LIN {X 0,Y 282.332,Z 323.54,A -85,B 0,C 180,E1 -17008.574,E2 -17008.574} C_VEL
LIN {X 0,Y 282.332,Z 323.54,A -85,B 0,C 180,E1 -17011.426,E2 -17011.426} C_VEL
LIN {X 0,Y 282.337,Z 322.95,A -85,B 0,C 180,E1 -17012.854,E2 -17012.854} C_VEL
LIN {X 0,Y 282.388,Z 320.499,A -85,B 0,C 180,E1 -17015.713,E2 -17015.713} C_VEL
LIN {X 0,Y 282.677,Z 317.547,A -85,B 0,C 180,E1 -17017.859,E2 -17017.859} C_VEL
LIN {X 0,Y 283.169,Z 313.557,A -85,B 0,C 180,E1 -17020.005,E2 -17020.005} C_VEL
LIN {X 0,Y 283.939,Z 308.424,A -85,B 0,C 180,E1 -17022.145,E2 -17022.145} C_VEL
LIN {X 0,Y 284.955,Z 303.165,A -85,B 0,C 180,E1 -17023.914,E2 -17023.914} C_VEL
LIN {X 0,Y 286.081,Z 296.847,A -85,B 0,C 180,E1 -17025.678,E2 -17025.678} C_VEL
LIN {X 0,Y 287.264,Z 290.899,A -85,B 0,C 180,E1 -17027.073,E2 -17027.073} C_VEL
LIN {X 0,Y 288.4,Z 283.969,A -85,B 0,C 180,E1 -17028.469,E2 -17028.469} C_VEL
LIN {X 0,Y 289.834,Z 275.791,A -85,B 0,C 180,E1 -17029.845,E2 -17029.845} C_VEL
LIN {X 0,Y 291.272,Z 267.283,A -85,B 0,C 180,E1 -17031.033,E2 -17031.033} C_VEL
LIN {X 0,Y 292.592,Z 258.569,A -85,B 0,C 180,E1 -17032.043,E2 -17032.043} C_VEL
LIN {X 0,Y 293.904,Z 248.813,A -85,B 0,C 180,E1 -17032.959,E2 -17032.959} C_VEL
LIN {X 0,Y 294.936,Z 240.021,A -85,B 0,C 180,E1 -17033.617,E2 -17033.617} C_VEL
LIN {X 0,Y 295.878,Z 230.095,A -85,B 0,C 180,E1 -17034.188,E2 -17034.188} C_VEL
LIN {X 0,Y 296.511,Z 220.239,A -85,B 0,C 180,E1 -17034.599,E2 -17034.599} C_VEL
LIN {X 0,Y 297.245,Z 197.417,A -85,B 0,C 180,E1 -17035.188,E2 -17035.188} C_VEL
LIN {X 0,Y 298.174,Z 158.869,A -85,B 0,C 180,E1 -17036.112,E2 -17036.112} C_VEL
LIN {X 0,Y 294.383,Z 137.525,A -85,B 0,C 180,E1 -17037.041,E2 -17037.041} C_VEL
LIN {X 0,Y 290.06,Z 118.484,A -85,B 0,C 180,E1 -17037.995,E2 -17037.995} C_VEL
LIN {X 0,Y 288.045,Z 112.98,A -85,B 0,C 180,E1 -17038.403,E2 -17038.403} C_VEL
LIN {X 0,Y 287.272,Z 108.749,A -85,B 0,C 180,E1 -17040.101,E2 -17040.101} C_VEL
LIN {X 0,Y 285.619,Z 100.449,A -85,B 0,C 180,E1 -17043.786,E2 -17043.786} C_VEL
LIN {X 0,Y 284.383,Z 94.573,A -85,B 0,C 180,E1 -17046.598,E2 -17046.598} C_VEL
LIN {X 0,Y 284.309,Z 94.538,A -85,B 0,C 180,E1 -17049.994,E2 -17049.994} C_VEL
LIN {X 0,Y 284.248,Z 94.574,A -85,B 0,C 180,E1 -17054.19,E2 -17054.19} C_VEL
LIN {X 0,Y 284.274,Z 94.574,A -85,B 0,C 180,E1 -17058.124,E2 -17058.124} C_VEL
LIN {X 0,Y 284.324,Z 94.568,A -85,B 0,C 180,E1 -17062.277,E2 -17062.277} C_VEL
LIN {X 0,Y 284.31,Z 94.547,A -85,B 0,C 180,E1 -17065.35,E2 -17065.35} C_VEL
LIN {X 0,Y 284.295,Z 94.571,A -85,B 0,C 180,E1 -17068.725,E2 -17068.725} C_VEL
LIN {X 0,Y 284.396,Z 94.53,A -85,B 0,C 180,E1 -17072.827,E2 -17072.827} C_VEL
LIN {X 0,Y 284.368,Z 94.562,A -85,B 0,C 180,E1 -17076.706,E2 -17076.706} C_VEL
LIN {X 0,Y 284.404,Z 94.52,A -85,B 0,C 180,E1 -17081.261,E2 -17081.261} C_VEL
LIN {X 0,Y 284.493,Z 94.54,A -85,B 0,C 180,E1 -17084.458,E2 -17084.458} C_VEL
LIN {X 0,Y 284.489,Z 94.522,A -85,B 0,C 180,E1 -17088.601,E2 -17088.601} C_VEL
LIN {X 0,Y 284.66,Z 94.494,A -85,B 0,C 180,E1 -17091.48,E2 -17091.48} C_VEL
LIN {X 0,Y 284.603,Z 94.533,A -85,B 0,C 180,E1 -17094.331,E2 -17094.331} C_VEL
LIN {X 0,Y 284.854,Z 94.474,A -85,B 0,C 180,E1 -17098.585,E2 -17098.585} C_VEL
LIN {X 0,Y 284.854,Z 94.471,A -85,B 0,C 180,E1 -17101.413,E2 -17101.413} C_VEL
LIN {X 0,Y 284.698,Z 94.51,A -85,B 0,C 180,E1 -17107.089,E2 -17107.089} C_VEL
LIN {X 0,Y 284.566,Z 94.499,A -85,B 0,C 180,E1 -17109.955,E2 -17109.955} C_VEL
LIN {X 0,Y 284.481,Z 94.548,A -85,B 0,C 180,E1 -17114.302,E2 -17114.302} C_VEL
LIN {X 0,Y 284.424,Z 94.535,A -85,B 0,C 180,E1 -17117.248,E2 -17117.248} C_VEL
LIN {X 0,Y 284.377,Z 94.535,A -85,B 0,C 180,E1 -17120.241,E2 -17120.241} C_VEL
LIN {X 0,Y 284.368,Z 94.561,A -85,B 0,C 180,E1 -17123.875,E2 -17123.875} C_VEL
LIN {X 0,Y 284.393,Z 94.532,A -85,B 0,C 180,E1 -17127.172,E2 -17127.172} C_VEL
LIN {X 0,Y 284.291,Z 94.573,A -85,B 0,C 180,E1 -17131.274,E2 -17131.274} C_VEL
LIN {X 0,Y 284.359,Z 94.546,A -85,B 0,C 180,E1 -17135.353,E2 -17135.353} C_VEL
LIN {X 0,Y 284.327,Z 94.57,A -85,B 0,C 180,E1 -17138.166,E2 -17138.166} C_VEL
LIN {X 0,Y 284.289,Z 94.564,A -85,B 0,C 180,E1 -17141.871,E2 -17141.871} C_VEL
LIN {X 0,Y 284.251,Z 94.537,A -85,B 0,C 180,E1 -17146.189,E2 -17146.189} C_VEL
LIN {X 0,Y 284.304,Z 94.538,A -85,B 0,C 180,E1 -17150.023,E2 -17150.023} C_VEL
LIN {X 0,Y 284.346,Z 94.545,A -85,B 0,C 180,E1 -17153.616,E2 -17153.616} C_VEL
LIN {X 0,Y 284.304,Z 94.553,A -85,B 0,C 180,E1 -17157.189,E2 -17157.189} C_VEL
LIN {X 0,Y 284.358,Z 94.704,A -85,B 0,C 180,E1 -17160.852,E2 -17160.852} C_VEL
LIN {X 0,Y 284.571,Z 95.611,A -85,B 0,C 180,E1 -17161.125,E2 -17161.125} C_VEL
LIN {X 0,Y 292.908,Z 111.214,A -85,B 0,C 180,E1 -17162.479,E2 -17162.479} C_VEL
LIN {X 0,Y 301.128,Z 122.682,A -85,B 0,C 180,E1 -17163.597,E2 -17163.597} C_VEL
LIN {X 0,Y 308.763,Z 131.233,A -85,B 0,C 180,E1 -17164.598,E2 -17164.598} C_VEL
LIN {X 0,Y 315.019,Z 137.865,A -85,B 0,C 180,E1 -17165.516,E2 -17165.516} C_VEL
LIN {X 0,Y 321.23,Z 144.234,A -85,B 0,C 180,E1 -17166.527,E2 -17166.527} C_VEL
LIN {X 0,Y 328.563,Z 151.312,A -85,B 0,C 180,E1 -17167.868,E2 -17167.868} C_VEL
LIN {X 0,Y 335.56,Z 157.924,A -85,B 0,C 180,E1 -17169.294,E2 -17169.294} C_VEL
LIN {X 0,Y 343.832,Z 165.121,A -85,B 0,C 180,E1 -17171.117,E2 -17171.117} C_VEL
LIN {X 0,Y 349.126,Z 169.383,A -85,B 0,C 180,E1 -17172.401,E2 -17172.401} C_VEL
LIN {X 0,Y 354.265,Z 173.621,A -85,B 0,C 180,E1 -17173.763,E2 -17173.763} C_VEL
LIN {X 0,Y 359.027,Z 177.249,A -85,B 0,C 180,E1 -17175.137,E2 -17175.137} C_VEL
LIN {X 0,Y 363.782,Z 181.091,A -85,B 0,C 180,E1 -17176.663,E2 -17176.663} C_VEL
LIN {X 0,Y 368.414,Z 183.996,A -85,B 0,C 180,E1 -17178.318,E2 -17178.318} C_VEL
LIN {X 0,Y 370.691,Z 185.609,A -85,B 0,C 180,E1 -17179.249,E2 -17179.249} C_VEL
LIN {X 0,Y 374.324,Z 188.697,A -85,B 0,C 180,E1 -17180.953,E2 -17180.953} C_VEL
LIN {X 0,Y 377.385,Z 190.784,A -85,B 0,C 180,E1 -17182.671,E2 -17182.671} C_VEL
LIN {X 0,Y 379.747,Z 192.052,A -85,B 0,C 180,E1 -17184.313,E2 -17184.313} C_VEL
LIN {X 0,Y 381.337,Z 192.728,A -85,B 0,C 180,E1 -17185.772,E2 -17185.772} C_VEL
LIN {X 0,Y 382.556,Z 193.147,A -85,B 0,C 180,E1 -17187.355,E2 -17187.355} C_VEL
LIN {X 0,Y 383.205,Z 193.6,A -85,B 0,C 180,E1 -17188.949,E2 -17188.949} C_VEL
LIN {X 0,Y 383.351,Z 193.507,A -85,B 0,C 180,E1 -17190,E2 -17190} C_VEL
LIN {X 0,Y 383.05,Z 193.43,A -85,B 0,C 180,E1 -17191.577,E2 -17191.577} C_VEL
LIN {X 0,Y 382.228,Z 192.953,A -85,B 0,C 180,E1 -17193.162,E2 -17193.162} C_VEL
LIN {X 0,Y 380.501,Z 192.419,A -85,B 0,C 180,E1 -17195.024,E2 -17195.024} C_VEL
LIN {X 0,Y 377.946,Z 191.113,A -85,B 0,C 180,E1 -17196.961,E2 -17196.961} C_VEL
LIN {X 0,Y 374.627,Z 188.924,A -85,B 0,C 180,E1 -17198.885,E2 -17198.885} C_VEL
LIN {X 0,Y 371.12,Z 186.009,A -85,B 0,C 180,E1 -17200.562,E2 -17200.562} C_VEL
LIN {X 0,Y 369.133,Z 184.402,A -85,B 0,C 180,E1 -17201.397,E2 -17201.397} C_VEL
LIN {X 0,Y 364.42,Z 181.507,A -85,B 0,C 180,E1 -17203.127,E2 -17203.127} C_VEL
LIN {X 0,Y 359.32,Z 177.506,A -85,B 0,C 180,E1 -17204.77,E2 -17204.77} C_VEL
LIN {X 0,Y 355.345,Z 174.403,A -85,B 0,C 180,E1 -17205.935,E2 -17205.935} C_VEL
LIN {X 0,Y 349.645,Z 169.914,A -85,B 0,C 180,E1 -17207.46,E2 -17207.46} C_VEL
LIN {X 0,Y 345.087,Z 166.059,A -85,B 0,C 180,E1 -17208.584,E2 -17208.584} C_VEL
LIN {X 0,Y 339.388,Z 161.216,A -85,B 0,C 180,E1 -17209.892,E2 -17209.892} C_VEL
LIN {X 0,Y 331.39,Z 154.073,A -85,B 0,C 180,E1 -17211.572,E2 -17211.572} C_VEL
LIN {X 0,Y 323.333,Z 146.328,A -85,B 0,C 180,E1 -17213.097,E2 -17213.097} C_VEL
LIN {X 0,Y 316.271,Z 139.268,A -85,B 0,C 180,E1 -17214.282,E2 -17214.282} C_VEL
LIN {X 0,Y 307.947,Z 130.457,A -85,B 0,C 180,E1 -17215.508,E2 -17215.508} C_VEL
LIN {X 0,Y 299.459,Z 120.55,A -85,B 0,C 180,E1 -17216.619,E2 -17216.619} C_VEL
LIN {X 0,Y 292.1,Z 109.823,A -85,B 0,C 180,E1 -17217.642,E2 -17217.642} C_VEL
LIN {X 0,Y 284.572,Z 95.609,A -85,B 0,C 180,E1 -17218.876,E2 -17218.876} C_VEL
LIN {X 0,Y 284.349,Z 94.626,A -85,B 0,C 180,E1 -17219.19,E2 -17219.19} C_VEL
LIN {X 0,Y 284.302,Z 94.55,A -85,B 0,C 180,E1 -17222.946,E2 -17222.946} C_VEL
LIN {X 0,Y 284.346,Z 94.544,A -85,B 0,C 180,E1 -17226.384,E2 -17226.384} C_VEL
LIN {X 0,Y 284.303,Z 94.538,A -85,B 0,C 180,E1 -17229.995,E2 -17229.995} C_VEL
LIN {X 0,Y 284.241,Z 94.546,A -85,B 0,C 180,E1 -17234.191,E2 -17234.191} C_VEL
LIN {X 0,Y 284.289,Z 94.564,A -85,B 0,C 180,E1 -17238.129,E2 -17238.129} C_VEL
LIN {X 0,Y 284.327,Z 94.57,A -85,B 0,C 180,E1 -17241.834,E2 -17241.834} C_VEL
LIN {X 0,Y 284.321,Z 94.547,A -85,B 0,C 180,E1 -17245.353,E2 -17245.353} C_VEL
LIN {X 0,Y 284.291,Z 94.573,A -85,B 0,C 180,E1 -17248.726,E2 -17248.726} C_VEL
LIN {X 0,Y 284.393,Z 94.532,A -85,B 0,C 180,E1 -17252.828,E2 -17252.828} C_VEL
LIN {X 0,Y 284.365,Z 94.565,A -85,B 0,C 180,E1 -17256.708,E2 -17256.708} C_VEL
LIN {X 0,Y 284.401,Z 94.525,A -85,B 0,C 180,E1 -17261.262,E2 -17261.262} C_VEL
LIN {X 0,Y 284.491,Z 94.544,A -85,B 0,C 180,E1 -17264.46,E2 -17264.46} C_VEL
LIN {X 0,Y 284.489,Z 94.522,A -85,B 0,C 180,E1 -17268.602,E2 -17268.602} C_VEL
LIN {X 0,Y 284.658,Z 94.497,A -85,B 0,C 180,E1 -17271.482,E2 -17271.482} C_VEL
LIN {X 0,Y 284.601,Z 94.533,A -85,B 0,C 180,E1 -17274.332,E2 -17274.332} C_VEL
LIN {X 0,Y 284.854,Z 94.471,A -85,B 0,C 180,E1 -17278.587,E2 -17278.587} C_VEL
LIN {X 0,Y 284.854,Z 94.474,A -85,B 0,C 180,E1 -17281.415,E2 -17281.415} C_VEL
LIN {X 0,Y 284.7,Z 94.508,A -85,B 0,C 180,E1 -17287.091,E2 -17287.091} C_VEL
LIN {X 0,Y 284.567,Z 94.498,A -85,B 0,C 180,E1 -17289.956,E2 -17289.956} C_VEL
LIN {X 0,Y 284.483,Z 94.545,A -85,B 0,C 180,E1 -17294.303,E2 -17294.303} C_VEL
LIN {X 0,Y 284.426,Z 94.529,A -85,B 0,C 180,E1 -17297.249,E2 -17297.249} C_VEL
LIN {X 0,Y 284.384,Z 94.531,A -85,B 0,C 180,E1 -17299.999,E2 -17299.999} C_VEL
LIN {X 0,Y 283.746,Z 94.627,A -85,B 0,C 180,E1 -17301.182,E2 -17301.182} C_VEL
LIN {X 0,Y 280.868,Z 94.998,A -85,B 0,C 180,E1 -17303.108,E2 -17303.108} C_VEL
LIN {X 0,Y 278.417,Z 95.294,A -85,B 0,C 180,E1 -17304.672,E2 -17304.672} C_VEL
LIN {X 0,Y 277.381,Z 95.409,A -85,B 0,C 180,E1 -17305.885,E2 -17305.885} C_VEL
LIN {X 0,Y 277.308,Z 95.414,A -85,B 0,C 180,E1 -17306.296,E2 -17306.296} C_VEL
LIN {X 0,Y 277.274,Z 95.446,A -85,B 0,C 180,E1 -17310.482,E2 -17310.482} C_VEL
LIN {X 0,Y 277.248,Z 95.426,A -85,B 0,C 180,E1 -17313.896,E2 -17313.896} C_VEL
LIN {X 0,Y 277.27,Z 95.447,A -85,B 0,C 180,E1 -17317.47,E2 -17317.47} C_VEL
LIN {X 0,Y 277.212,Z 95.444,A -85,B 0,C 180,E1 -17321.237,E2 -17321.237} C_VEL
LIN {X 0,Y 277.203,Z 95.446,A -85,B 0,C 180,E1 -17325.227,E2 -17325.227} C_VEL
LIN {X 0,Y 277.225,Z 95.42,A -85,B 0,C 180,E1 -17329.513,E2 -17329.513} C_VEL
LIN {X 0,Y 277.341,Z 95.56,A -85,B 0,C 180,E1 -17332.959,E2 -17332.959} C_VEL
LIN {X 0,Y 278.814,Z 102.621,A -85,B 0,C 180,E1 -17336.32,E2 -17336.32} C_VEL
LIN {X 0,Y 280.364,Z 110.466,A -85,B 0,C 180,E1 -17339.911,E2 -17339.911} C_VEL
LIN {X 0,Y 280.827,Z 112.758,A -85,B 0,C 180,E1 -17340.794,E2 -17340.794} C_VEL
LIN {X 0,Y 284.469,Z 122.35,A -85,B 0,C 180,E1 -17341.518,E2 -17341.518} C_VEL
LIN {X 0,Y 289.627,Z 146.77,A -85,B 0,C 180,E1 -17342.734,E2 -17342.734} C_VEL
LIN {X 0,Y 291.872,Z 160.971,A -85,B 0,C 180,E1 -17343.342,E2 -17343.342} C_VEL
LIN {X 0,Y 290.223,Z 218.73,A -85,B 0,C 180,E1 -17344.783,E2 -17344.783} C_VEL
LIN {X 0,Y 289.49,Z 229.031,A -85,B 0,C 180,E1 -17345.195,E2 -17345.195} C_VEL
LIN {X 0,Y 288.543,Z 238.542,A -85,B 0,C 180,E1 -17345.731,E2 -17345.731} C_VEL
LIN {X 0,Y 287.418,Z 248.624,A -85,B 0,C 180,E1 -17346.492,E2 -17346.492} C_VEL
LIN {X 0,Y 286.034,Z 258.379,A -85,B 0,C 180,E1 -17347.424,E2 -17347.424} C_VEL
LIN {X 0,Y 284.398,Z 268.442,A -85,B 0,C 180,E1 -17348.623,E2 -17348.623} C_VEL
LIN {X 0,Y 282.361,Z 279.94,A -85,B 0,C 180,E1 -17350.366,E2 -17350.366} C_VEL
LIN {X 0,Y 280.716,Z 288.731,A -85,B 0,C 180,E1 -17352.06,E2 -17352.06} C_VEL
LIN {X 0,Y 279.503,Z 295.28,A -85,B 0,C 180,E1 -17353.568,E2 -17353.568} C_VEL
LIN {X 0,Y 278.263,Z 301.818,A -85,B 0,C 180,E1 -17355.371,E2 -17355.371} C_VEL
LIN {X 0,Y 277.338,Z 306.317,A -85,B 0,C 180,E1 -17356.817,E2 -17356.817} C_VEL
LIN {X 0,Y 276.386,Z 311.811,A -85,B 0,C 180,E1 -17359.006,E2 -17359.006} C_VEL
LIN {X 0,Y 275.745,Z 316.138,A -85,B 0,C 180,E1 -17361.204,E2 -17361.204} C_VEL
LIN {X 0,Y 275.496,Z 318.507,A -85,B 0,C 180,E1 -17362.672,E2 -17362.672} C_VEL
LIN {X 0,Y 275.249,Z 321,A -85,B 0,C 180,E1 -17364.751,E2 -17364.751} C_VEL
LIN {X 0,Y 275.246,Z 322.759,A -85,B 0,C 180,E1 -17367.073,E2 -17367.073} C_VEL
LIN {X 0,Y 275.256,Z 323.35,A -85,B 0,C 180,E1 -17368.537,E2 -17368.537} C_VEL
LIN {X 0,Y 275.256,Z 323.35,A -85,B 0,C 180,E1 -17371.463,E2 -17371.463} C_VEL
LIN {X 0,Y 275.246,Z 322.759,A -85,B 0,C 180,E1 -17372.927,E2 -17372.927} C_VEL
LIN {X 0,Y 275.302,Z 320.308,A -85,B 0,C 180,E1 -17375.861,E2 -17375.861} C_VEL
LIN {X 0,Y 275.606,Z 317.356,A -85,B 0,C 180,E1 -17378.062,E2 -17378.062} C_VEL
LIN {X 0,Y 276.159,Z 313.366,A -85,B 0,C 180,E1 -17380.262,E2 -17380.262} C_VEL
LIN {X 0,Y 276.965,Z 308.233,A -85,B 0,C 180,E1 -17382.456,E2 -17382.456} C_VEL
LIN {X 0,Y 278.02,Z 302.973,A -85,B 0,C 180,E1 -17384.269,E2 -17384.269} C_VEL
LIN {X 0,Y 279.218,Z 296.655,A -85,B 0,C 180,E1 -17386.074,E2 -17386.074} C_VEL
LIN {X 0,Y 280.673,Z 289.683,A -85,B 0,C 180,E1 -17387.723,E2 -17387.723} C_VEL
LIN {X 0,Y 281.661,Z 283.778,A -85,B 0,C 180,E1 -17388.928,E2 -17388.928} C_VEL
LIN {X 0,Y 283.156,Z 275.601,A -85,B 0,C 180,E1 -17390.333,E2 -17390.333} C_VEL
LIN {X 0,Y 284.652,Z 267.092,A -85,B 0,C 180,E1 -17391.547,E2 -17391.547} C_VEL
LIN {X 0,Y 286.016,Z 258.378,A -85,B 0,C 180,E1 -17392.578,E2 -17392.578} C_VEL
LIN {X 0,Y 287.379,Z 248.622,A -85,B 0,C 180,E1 -17393.511,E2 -17393.511} C_VEL
LIN {X 0,Y 288.438,Z 239.831,A -85,B 0,C 180,E1 -17394.183,E2 -17394.183} C_VEL
LIN {X 0,Y 289.418,Z 229.905,A -85,B 0,C 180,E1 -17394.764,E2 -17394.764} C_VEL
LIN {X 0,Y 290.084,Z 220.049,A -85,B 0,C 180,E1 -17395.182,E2 -17395.182} C_VEL
LIN {X 0,Y 290.824,Z 197.226,A -85,B 0,C 180,E1 -17395.784,E2 -17395.784} C_VEL
LIN {X 0,Y 291.8,Z 159.943,A -85,B 0,C 180,E1 -17396.693,E2 -17396.693} C_VEL
LIN {X 0,Y 288.2,Z 139.453,A -85,B 0,C 180,E1 -17397.612,E2 -17397.612} C_VEL
LIN {X 0,Y 284.11,Z 121.147,A -85,B 0,C 180,E1 -17398.555,E2 -17398.555} C_VEL
LIN {X 0,Y 280.821,Z 112.765,A -85,B 0,C 180,E1 -17399.203,E2 -17399.203} C_VEL
LIN {X 0,Y 280.099,Z 109.079,A -85,B 0,C 180,E1 -17400.721,E2 -17400.721} C_VEL
LIN {X 0,Y 278.839,Z 102.522,A -85,B 0,C 180,E1 -17403.72,E2 -17403.72} C_VEL
LIN {X 0,Y 277.342,Z 95.462,A -85,B 0,C 180,E1 -17407.144,E2 -17407.144} C_VEL
LIN {X 0,Y 277.212,Z 95.428,A -85,B 0,C 180,E1 -17411.236,E2 -17411.236} C_VEL
LIN {X 0,Y 277.203,Z 95.446,A -85,B 0,C 180,E1 -17415.226,E2 -17415.226} C_VEL
LIN {X 0,Y 277.224,Z 95.437,A -85,B 0,C 180,E1 -17419.512,E2 -17419.512} C_VEL
LIN {X 0,Y 277.27,Z 95.447,A -85,B 0,C 180,E1 -17422.53,E2 -17422.53} C_VEL
LIN {X 0,Y 277.248,Z 95.426,A -85,B 0,C 180,E1 -17426.104,E2 -17426.104} C_VEL
LIN {X 0,Y 277.263,Z 95.447,A -85,B 0,C 180,E1 -17429.538,E2 -17429.538} C_VEL
LIN {X 0,Y 277.358,Z 95.406,A -85,B 0,C 180,E1 -17432.863,E2 -17432.863} C_VEL
LIN {X 0,Y 277.33,Z 95.435,A -85,B 0,C 180,E1 -17436.079,E2 -17436.079} C_VEL
LIN {X 0,Y 277.346,Z 95.4,A -85,B 0,C 180,E1 -17440.765,E2 -17440.765} C_VEL
LIN {X 0,Y 277.436,Z 95.423,A -85,B 0,C 180,E1 -17445.325,E2 -17445.325} C_VEL
LIN {X 0,Y 277.507,Z 95.378,A -85,B 0,C 180,E1 -17449.788,E2 -17449.788} C_VEL
LIN {X 0,Y 277.655,Z 95.382,A -85,B 0,C 180,E1 -17452.728,E2 -17452.728} C_VEL
LIN {X 0,Y 277.82,Z 95.35,A -85,B 0,C 180,E1 -17458.55,E2 -17458.55} C_VEL
LIN {X 0,Y 277.82,Z 95.347,A -85,B 0,C 180,E1 -17461.449,E2 -17461.449} C_VEL
LIN {X 0,Y 277.653,Z 95.384,A -85,B 0,C 180,E1 -17467.27,E2 -17467.27} C_VEL
LIN {X 0,Y 277.507,Z 95.379,A -85,B 0,C 180,E1 -17470.21,E2 -17470.21} C_VEL
LIN {X 0,Y 277.434,Z 95.426,A -85,B 0,C 180,E1 -17474.673,E2 -17474.673} C_VEL
LIN {X 0,Y 277.343,Z 95.403,A -85,B 0,C 180,E1 -17479.233,E2 -17479.233} C_VEL
LIN {X 0,Y 277.318,Z 95.439,A -85,B 0,C 180,E1 -17484.17,E2 -17484.17} C_VEL
LIN {X 0,Y 277.321,Z 95.412,A -85,B 0,C 180,E1 -17487.504,E2 -17487.504} C_VEL
LIN {X 0,Y 277.27,Z 95.446,A -85,B 0,C 180,E1 -17490.481,E2 -17490.481} C_VEL
LIN {X 0,Y 277.251,Z 95.428,A -85,B 0,C 180,E1 -17493.894,E2 -17493.894} C_VEL
LIN {X 0,Y 277.283,Z 95.447,A -85,B 0,C 180,E1 -17497.466,E2 -17497.466} C_VEL
LIN {X 0,Y 277.231,Z 95.436,A -85,B 0,C 180,E1 -17501.232,E2 -17501.232} C_VEL
LIN {X 0,Y 277.2,Z 95.434,A -85,B 0,C 180,E1 -17505.225,E2 -17505.225} C_VEL
LIN {X 0,Y 277.218,Z 95.409,A -85,B 0,C 180,E1 -17509.512,E2 -17509.512} C_VEL
LIN {X 0,Y 277.278,Z 95.445,A -85,B 0,C 180,E1 -17512.533,E2 -17512.533} C_VEL
LIN {X 0,Y 277.25,Z 95.415,A -85,B 0,C 180,E1 -17516.105,E2 -17516.105} C_VEL
LIN {X 0,Y 277.307,Z 95.57,A -85,B 0,C 180,E1 -17520.071,E2 -17520.071} C_VEL
LIN {X 0,Y 277.558,Z 96.523,A -85,B 0,C 180,E1 -17520.347,E2 -17520.347} C_VEL
LIN {X 0,Y 287.675,Z 115.487,A -85,B 0,C 180,E1 -17522.049,E2 -17522.049} C_VEL
LIN {X 0,Y 296.033,Z 127.245,A -85,B 0,C 180,E1 -17523.224,E2 -17523.224} C_VEL
LIN {X 0,Y 304.437,Z 136.633,A -85,B 0,C 180,E1 -17524.285,E2 -17524.285} C_VEL
LIN {X 0,Y 311.55,Z 144.001,A -85,B 0,C 180,E1 -17525.264,E2 -17525.264} C_VEL
LIN {X 0,Y 317.642,Z 150.071,A -85,B 0,C 180,E1 -17526.194,E2 -17526.194} C_VEL
LIN {X 0,Y 324.32,Z 156.446,A -85,B 0,C 180,E1 -17527.349,E2 -17527.349} C_VEL
LIN {X 0,Y 332.199,Z 163.7,A -85,B 0,C 180,E1 -17528.859,E2 -17528.859} C_VEL
LIN {X 0,Y 340.746,Z 171.076,A -85,B 0,C 180,E1 -17530.692,E2 -17530.692} C_VEL
LIN {X 0,Y 346.717,Z 175.77,A -85,B 0,C 180,E1 -17532.086,E2 -17532.086} C_VEL
LIN {X 0,Y 352.189,Z 180.199,A -85,B 0,C 180,E1 -17533.491,E2 -17533.491} C_VEL
LIN {X 0,Y 357.449,Z 184.156,A -85,B 0,C 180,E1 -17534.97,E2 -17534.97} C_VEL
LIN {X 0,Y 362.886,Z 188.383,A -85,B 0,C 180,E1 -17536.697,E2 -17536.697} C_VEL
LIN {X 0,Y 367.765,Z 191.274,A -85,B 0,C 180,E1 -17538.433,E2 -17538.433} C_VEL
LIN {X 0,Y 372.315,Z 195.056,A -85,B 0,C 180,E1 -17540.433,E2 -17540.433} C_VEL
LIN {X 0,Y 375.651,Z 197.365,A -85,B 0,C 180,E1 -17542.185,E2 -17542.185} C_VEL
LIN {X 0,Y 378.536,Z 198.953,A -85,B 0,C 180,E1 -17544.075,E2 -17544.075} C_VEL
LIN {X 0,Y 380.515,Z 199.785,A -85,B 0,C 180,E1 -17545.828,E2 -17545.828} C_VEL
LIN {X 0,Y 381.686,Z 200.194,A -85,B 0,C 180,E1 -17547.349,E2 -17547.349} C_VEL
LIN {X 0,Y 382.34,Z 200.646,A -85,B 0,C 180,E1 -17548.947,E2 -17548.947} C_VEL
LIN {X 0,Y 382.488,Z 200.539,A -85,B 0,C 180,E1 -17550,E2 -17550} C_VEL
LIN {X 0,Y 382.181,Z 200.478,A -85,B 0,C 180,E1 -17551.581,E2 -17551.581} C_VEL
LIN {X 0,Y 381.092,Z 199.929,A -85,B 0,C 180,E1 -17553.513,E2 -17553.513} C_VEL
LIN {X 0,Y 379.107,Z 199.217,A -85,B 0,C 180,E1 -17555.477,E2 -17555.477} C_VEL
LIN {X 0,Y 376.465,Z 197.808,A -85,B 0,C 180,E1 -17557.348,E2 -17557.348} C_VEL
LIN {X 0,Y 373.181,Z 195.688,A -85,B 0,C 180,E1 -17559.153,E2 -17559.153} C_VEL
LIN {X 0,Y 369.493,Z 192.66,A -85,B 0,C 180,E1 -17560.852,E2 -17560.852} C_VEL
LIN {X 0,Y 367.139,Z 190.928,A -85,B 0,C 180,E1 -17561.798,E2 -17561.798} C_VEL
LIN {X 0,Y 362.576,Z 188.136,A -85,B 0,C 180,E1 -17563.407,E2 -17563.407} C_VEL
LIN {X 0,Y 357.452,Z 184.132,A -85,B 0,C 180,E1 -17565.03,E2 -17565.03} C_VEL
LIN {X 0,Y 351.476,Z 179.651,A -85,B 0,C 180,E1 -17566.701,E2 -17566.701} C_VEL
LIN {X 0,Y 345.974,Z 175.162,A -85,B 0,C 180,E1 -17568.096,E2 -17568.096} C_VEL
LIN {X 0,Y 337.981,Z 168.729,A -85,B 0,C 180,E1 -17569.928,E2 -17569.928} C_VEL
LIN {X 0,Y 329.178,Z 160.994,A -85,B 0,C 180,E1 -17571.739,E2 -17571.739} C_VEL
LIN {X 0,Y 320.365,Z 152.707,A -85,B 0,C 180,E1 -17573.351,E2 -17573.351} C_VEL
LIN {X 0,Y 312.398,Z 144.958,A -85,B 0,C 180,E1 -17574.611,E2 -17574.611} C_VEL
LIN {X 0,Y 303.796,Z 136.018,A -85,B 0,C 180,E1 -17575.795,E2 -17575.795} C_VEL
LIN {X 0,Y 294.334,Z 125.049,A -85,B 0,C 180,E1 -17577.003,E2 -17577.003} C_VEL
LIN {X 0,Y 287.007,Z 114.312,A -85,B 0,C 180,E1 -17578.055,E2 -17578.055} C_VEL
LIN {X 0,Y 277.551,Z 96.544,A -85,B 0,C 180,E1 -17579.65,E2 -17579.65} C_VEL
LIN {X 0,Y 277.302,Z 95.517,A -85,B 0,C 180,E1 -17579.965,E2 -17579.965} C_VEL
LIN {X 0,Y 277.251,Z 95.415,A -85,B 0,C 180,E1 -17583.895,E2 -17583.895} C_VEL
LIN {X 0,Y 277.278,Z 95.445,A -85,B 0,C 180,E1 -17587.467,E2 -17587.467} C_VEL
LIN {X 0,Y 277.206,Z 95.401,A -85,B 0,C 180,E1 -17591.237,E2 -17591.237} C_VEL
LIN {X 0,Y 277.204,Z 95.445,A -85,B 0,C 180,E1 -17595.226,E2 -17595.226} C_VEL
LIN {X 0,Y 277.257,Z 95.431,A -85,B 0,C 180,E1 -17599.504,E2 -17599.504} C_VEL
LIN {X 0,Y 277.283,Z 95.447,A -85,B 0,C 180,E1 -17602.534,E2 -17602.534} C_VEL
LIN {X 0,Y 277.251,Z 95.428,A -85,B 0,C 180,E1 -17606.106,E2 -17606.106} C_VEL
LIN {X 0,Y 277.259,Z 95.448,A -85,B 0,C 180,E1 -17609.539,E2 -17609.539} C_VEL
LIN {X 0,Y 277.355,Z 95.408,A -85,B 0,C 180,E1 -17612.865,E2 -17612.865} C_VEL
LIN {X 0,Y 277.327,Z 95.438,A -85,B 0,C 180,E1 -17616.08,E2 -17616.08} C_VEL
LIN {X 0,Y 277.343,Z 95.403,A -85,B 0,C 180,E1 -17620.767,E2 -17620.767} C_VEL
LIN {X 0,Y 277.434,Z 95.426,A -85,B 0,C 180,E1 -17625.327,E2 -17625.327} C_VEL
LIN {X 0,Y 277.507,Z 95.379,A -85,B 0,C 180,E1 -17629.79,E2 -17629.79} C_VEL
LIN {X 0,Y 277.653,Z 95.384,A -85,B 0,C 180,E1 -17632.73,E2 -17632.73} C_VEL
LIN {X 0,Y 277.82,Z 95.347,A -85,B 0,C 180,E1 -17638.551,E2 -17638.551} C_VEL
LIN {X 0,Y 277.82,Z 95.35,A -85,B 0,C 180,E1 -17641.45,E2 -17641.45} C_VEL
LIN {X 0,Y 277.655,Z 95.382,A -85,B 0,C 180,E1 -17647.272,E2 -17647.272} C_VEL
LIN {X 0,Y 277.507,Z 95.378,A -85,B 0,C 180,E1 -17650.212,E2 -17650.212} C_VEL
LIN {X 0,Y 277.436,Z 95.423,A -85,B 0,C 180,E1 -17654.675,E2 -17654.675} C_VEL
LIN {X 0,Y 277.346,Z 95.4,A -85,B 0,C 180,E1 -17659.235,E2 -17659.235} C_VEL
LIN {X 0,Y 277.321,Z 95.435,A -85,B 0,C 180,E1 -17664.171,E2 -17664.171} C_VEL
LIN {X 0,Y 277.308,Z 95.414,A -85,B 0,C 180,E1 -17666.296,E2 -17666.296} C_VEL
LIN {X 0,Y 276.647,Z 95.498,A -85,B 0,C 180,E1 -17667.508,E2 -17667.508} C_VEL
LIN {X 0,Y 273.73,Z 95.881,A -85,B 0,C 180,E1 -17669.48,E2 -17669.48} C_VEL
LIN {X 0,Y 271.265,Z 96.196,A -85,B 0,C 180,E1 -17671.083,E2 -17671.083} C_VEL
LIN {X 0,Y 270.243,Z 96.313,A -85,B 0,C 180,E1 -17672.327,E2 -17672.327} C_VEL
LIN {X 0,Y 270.18,Z 96.312,A -85,B 0,C 180,E1 -17672.749,E2 -17672.749} C_VEL
LIN {X 0,Y 270.219,Z 96.323,A -85,B 0,C 180,E1 -17676.742,E2 -17676.742} C_VEL
LIN {X 0,Y 270.171,Z 96.318,A -85,B 0,C 180,E1 -17681.029,E2 -17681.029} C_VEL
LIN {X 0,Y 270.154,Z 96.324,A -85,B 0,C 180,E1 -17685.38,E2 -17685.38} C_VEL
LIN {X 0,Y 270.176,Z 96.298,A -85,B 0,C 180,E1 -17689.435,E2 -17689.435} C_VEL
LIN {X 0,Y 270.287,Z 96.444,A -85,B 0,C 180,E1 -17692.335,E2 -17692.335} C_VEL
LIN {X 0,Y 271.787,Z 103.543,A -85,B 0,C 180,E1 -17695.841,E2 -17695.841} C_VEL
LIN {X 0,Y 273.526,Z 112.348,A -85,B 0,C 180,E1 -17699.902,E2 -17699.902} C_VEL
LIN {X 0,Y 275.126,Z 116.309,A -85,B 0,C 180,E1 -17700.288,E2 -17700.288} C_VEL
LIN {X 0,Y 278.61,Z 125.322,A -85,B 0,C 180,E1 -17700.953,E2 -17700.953} C_VEL
LIN {X 0,Y 283.388,Z 148.392,A -85,B 0,C 180,E1 -17702.133,E2 -17702.133} C_VEL
LIN {X 0,Y 285.505,Z 161.817,A -85,B 0,C 180,E1 -17702.728,E2 -17702.728} C_VEL
LIN {X 0,Y 283.824,Z 218.546,A -85,B 0,C 180,E1 -17704.173,E2 -17704.173} C_VEL
LIN {X 0,Y 283.076,Z 228.841,A -85,B 0,C 180,E1 -17704.593,E2 -17704.593} C_VEL
LIN {X 0,Y 282.104,Z 238.352,A -85,B 0,C 180,E1 -17705.14,E2 -17705.14} C_VEL
LIN {X 0,Y 281.03,Z 247.426,A -85,B 0,C 180,E1 -17705.826,E2 -17705.826} C_VEL
LIN {X 0,Y 279.698,Z 256.556,A -85,B 0,C 180,E1 -17706.687,E2 -17706.687} C_VEL
LIN {X 0,Y 278.269,Z 265.55,A -85,B 0,C 180,E1 -17707.738,E2 -17707.738} C_VEL
LIN {X 0,Y 276.701,Z 274.275,A -85,B 0,C 180,E1 -17708.976,E2 -17708.976} C_VEL
LIN {X 0,Y 275.276,Z 281.667,A -85,B 0,C 180,E1 -17710.228,E2 -17710.228} C_VEL
LIN {X 0,Y 273.809,Z 289.215,A -85,B 0,C 180,E1 -17711.752,E2 -17711.752} C_VEL
LIN {X 0,Y 272.688,Z 295.089,A -85,B 0,C 180,E1 -17713.145,E2 -17713.145} C_VEL
LIN {X 0,Y 271.385,Z 301.627,A -85,B 0,C 180,E1 -17714.991,E2 -17714.991} C_VEL
LIN {X 0,Y 270.412,Z 306.126,A -85,B 0,C 180,E1 -17716.473,E2 -17716.473} C_VEL
LIN {X 0,Y 269.381,Z 311.619,A -85,B 0,C 180,E1 -17718.716,E2 -17718.716} C_VEL
LIN {X 0,Y 268.707,Z 315.946,A -85,B 0,C 180,E1 -17720.971,E2 -17720.971} C_VEL
LIN {X 0,Y 268.418,Z 318.316,A -85,B 0,C 180,E1 -17722.478,E2 -17722.478} C_VEL
LIN {X 0,Y 268.158,Z 320.986,A -85,B 0,C 180,E1 -17724.831,E2 -17724.831} C_VEL
LIN {X 0,Y 268.157,Z 322.569,A -85,B 0,C 180,E1 -17726.995,E2 -17726.995} C_VEL
LIN {X 0,Y 268.182,Z 323.16,A -85,B 0,C 180,E1 -17728.498,E2 -17728.498} C_VEL
LIN {X 0,Y 268.182,Z 323.16,A -85,B 0,C 180,E1 -17731.502,E2 -17731.502} C_VEL
LIN {X 0,Y 268.157,Z 322.569,A -85,B 0,C 180,E1 -17733.005,E2 -17733.005} C_VEL
LIN {X 0,Y 268.227,Z 320.117,A -85,B 0,C 180,E1 -17736.016,E2 -17736.016} C_VEL
LIN {X 0,Y 268.548,Z 317.164,A -85,B 0,C 180,E1 -17738.276,E2 -17738.276} C_VEL
LIN {X 0,Y 269.141,Z 313.174,A -85,B 0,C 180,E1 -17740.532,E2 -17740.532} C_VEL
LIN {X 0,Y 270.009,Z 308.042,A -85,B 0,C 180,E1 -17742.782,E2 -17742.782} C_VEL
LIN {X 0,Y 271.115,Z 302.781,A -85,B 0,C 180,E1 -17744.64,E2 -17744.64} C_VEL
LIN {X 0,Y 272.381,Z 296.464,A -85,B 0,C 180,E1 -17746.488,E2 -17746.488} C_VEL
LIN {X 0,Y 273.664,Z 290.516,A -85,B 0,C 180,E1 -17747.949,E2 -17747.949} C_VEL
LIN {X 0,Y 274.928,Z 283.587,A -85,B 0,C 180,E1 -17749.41,E2 -17749.41} C_VEL
LIN {X 0,Y 276.496,Z 275.41,A -85,B 0,C 180,E1 -17750.846,E2 -17750.846} C_VEL
LIN {X 0,Y 278.042,Z 266.901,A -85,B 0,C 180,E1 -17752.086,E2 -17752.086} C_VEL
LIN {X 0,Y 279.477,Z 258.188,A -85,B 0,C 180,E1 -17753.136,E2 -17753.136} C_VEL
LIN {X 0,Y 280.888,Z 248.432,A -85,B 0,C 180,E1 -17754.089,E2 -17754.089} C_VEL
LIN {X 0,Y 281.964,Z 239.64,A -85,B 0,C 180,E1 -17754.775,E2 -17754.775} C_VEL
LIN {X 0,Y 282.988,Z 229.714,A -85,B 0,C 180,E1 -17755.366,E2 -17755.366} C_VEL
LIN {X 0,Y 283.687,Z 219.859,A -85,B 0,C 180,E1 -17755.791,E2 -17755.791} C_VEL
LIN {X 0,Y 284.449,Z 197.036,A -85,B 0,C 180,E1 -17756.406,E2 -17756.406} C_VEL
LIN {X 0,Y 285.392,Z 160.584,A -85,B 0,C 180,E1 -17757.318,E2 -17757.318} C_VEL
LIN {X 0,Y 281.859,Z 140.46,A -85,B 0,C 180,E1 -17758.254,E2 -17758.254} C_VEL
LIN {X 0,Y 278.13,Z 123.7,A -85,B 0,C 180,E1 -17759.148,E2 -17759.148} C_VEL
LIN {X 0,Y 273.649,Z 112.769,A -85,B 0,C 180,E1 -17760.021,E2 -17760.021} C_VEL
LIN {X 0,Y 273.457,Z 111.921,A -85,B 0,C 180,E1 -17760.232,E2 -17760.232} C_VEL
LIN {X 0,Y 271.811,Z 103.519,A -85,B 0,C 180,E1 -17764.166,E2 -17764.166} C_VEL
LIN {X 0,Y 270.283,Z 96.383,A -85,B 0,C 180,E1 -17767.724,E2 -17767.724} C_VEL
LIN {X 0,Y 270.174,Z 96.326,A -85,B 0,C 180,E1 -17772.558,E2 -17772.558} C_VEL
LIN {X 0,Y 270.167,Z 96.332,A -85,B 0,C 180,E1 -17776.75,E2 -17776.75} C_VEL
LIN {X 0,Y 270.175,Z 96.315,A -85,B 0,C 180,E1 -17779.433,E2 -17779.433} C_VEL
LIN {X 0,Y 270.228,Z 96.319,A -85,B 0,C 180,E1 -17783.73,E2 -17783.73} C_VEL
LIN {X 0,Y 270.204,Z 96.308,A -85,B 0,C 180,E1 -17786.892,E2 -17786.892} C_VEL
LIN {X 0,Y 270.197,Z 96.323,A -85,B 0,C 180,E1 -17790.382,E2 -17790.382} C_VEL
LIN {X 0,Y 270.264,Z 96.292,A -85,B 0,C 180,E1 -17793.763,E2 -17793.763} C_VEL
LIN {X 0,Y 270.235,Z 96.322,A -85,B 0,C 180,E1 -17797.038,E2 -17797.038} C_VEL
LIN {X 0,Y 270.303,Z 96.28,A -85,B 0,C 180,E1 -17800.244,E2 -17800.244} C_VEL
LIN {X 0,Y 270.404,Z 96.3,A -85,B 0,C 180,E1 -17804.935,E2 -17804.935} C_VEL
LIN {X 0,Y 270.442,Z 96.258,A -85,B 0,C 180,E1 -17809.518,E2 -17809.518} C_VEL
LIN {X 0,Y 270.613,Z 96.255,A -85,B 0,C 180,E1 -17812.538,E2 -17812.538} C_VEL
LIN {X 0,Y 270.786,Z 96.225,A -85,B 0,C 180,E1 -17818.512,E2 -17818.512} C_VEL
LIN {X 0,Y 270.786,Z 96.222,A -85,B 0,C 180,E1 -17821.486,E2 -17821.486} C_VEL
LIN {X 0,Y 270.611,Z 96.258,A -85,B 0,C 180,E1 -17827.46,E2 -17827.46} C_VEL
LIN {X 0,Y 270.442,Z 96.259,A -85,B 0,C 180,E1 -17830.48,E2 -17830.48} C_VEL
LIN {X 0,Y 270.402,Z 96.304,A -85,B 0,C 180,E1 -17835.064,E2 -17835.064} C_VEL
LIN {X 0,Y 270.3,Z 96.282,A -85,B 0,C 180,E1 -17839.755,E2 -17839.755} C_VEL
LIN {X 0,Y 270.272,Z 96.314,A -85,B 0,C 180,E1 -17844.585,E2 -17844.585} C_VEL
LIN {X 0,Y 270.268,Z 96.292,A -85,B 0,C 180,E1 -17847.908,E2 -17847.908} C_VEL
LIN {X 0,Y 270.182,Z 96.331,A -85,B 0,C 180,E1 -17851.347,E2 -17851.347} C_VEL
LIN {X 0,Y 270.213,Z 96.304,A -85,B 0,C 180,E1 -17854.903,E2 -17854.903} C_VEL
LIN {X 0,Y 270.22,Z 96.321,A -85,B 0,C 180,E1 -17858.716,E2 -17858.716} C_VEL
LIN {X 0,Y 270.181,Z 96.327,A -85,B 0,C 180,E1 -17862.555,E2 -17862.555} C_VEL
LIN {X 0,Y 270.161,Z 96.281,A -85,B 0,C 180,E1 -17866.751,E2 -17866.751} C_VEL
LIN {X 0,Y 270.219,Z 96.32,A -85,B 0,C 180,E1 -17871.283,E2 -17871.283} C_VEL
LIN {X 0,Y 270.211,Z 96.288,A -85,B 0,C 180,E1 -17875.096,E2 -17875.096} C_VEL
LIN {X 0,Y 270.244,Z 96.553,A -85,B 0,C 180,E1 -17879.299,E2 -17879.299} C_VEL
LIN {X 0,Y 270.53,Z 97.62,A -85,B 0,C 180,E1 -17879.534,E2 -17879.534} C_VEL
LIN {X 0,Y 282.82,Z 120.333,A -85,B 0,C 180,E1 -17881.659,E2 -17881.659} C_VEL
LIN {X 0,Y 291.434,Z 132.405,A -85,B 0,C 180,E1 -17882.904,E2 -17882.904} C_VEL
LIN {X 0,Y 302.649,Z 144.837,A -85,B 0,C 180,E1 -17884.325,E2 -17884.325} C_VEL
LIN {X 0,Y 312.028,Z 154.153,A -85,B 0,C 180,E1 -17885.596,E2 -17885.596} C_VEL
LIN {X 0,Y 320.553,Z 162.057,A -85,B 0,C 180,E1 -17886.94,E2 -17886.94} C_VEL
LIN {X 0,Y 329.27,Z 169.9,A -85,B 0,C 180,E1 -17888.54,E2 -17888.54} C_VEL
LIN {X 0,Y 338.275,Z 177.506,A -85,B 0,C 180,E1 -17890.407,E2 -17890.407} C_VEL
LIN {X 0,Y 343.951,Z 181.912,A -85,B 0,C 180,E1 -17891.701,E2 -17891.701} C_VEL
LIN {X 0,Y 349.66,Z 186.511,A -85,B 0,C 180,E1 -17893.119,E2 -17893.119} C_VEL
LIN {X 0,Y 355.428,Z 190.732,A -85,B 0,C 180,E1 -17894.682,E2 -17894.682} C_VEL
LIN {X 0,Y 361.296,Z 195.19,A -85,B 0,C 180,E1 -17896.501,E2 -17896.501} C_VEL
LIN {X 0,Y 366.307,Z 198.126,A -85,B 0,C 180,E1 -17898.249,E2 -17898.249} C_VEL
LIN {X 0,Y 370.879,Z 201.816,A -85,B 0,C 180,E1 -17900.186,E2 -17900.186} C_VEL
LIN {X 0,Y 374.242,Z 204.145,A -85,B 0,C 180,E1 -17901.892,E2 -17901.892} C_VEL
LIN {X 0,Y 377.191,Z 205.795,A -85,B 0,C 180,E1 -17903.737,E2 -17903.737} C_VEL
LIN {X 0,Y 379.566,Z 206.803,A -85,B 0,C 180,E1 -17905.753,E2 -17905.753} C_VEL
LIN {X 0,Y 380.815,Z 207.242,A -85,B 0,C 180,E1 -17907.343,E2 -17907.343} C_VEL
LIN {X 0,Y 381.474,Z 207.692,A -85,B 0,C 180,E1 -17908.944,E2 -17908.944} C_VEL
LIN {X 0,Y 381.624,Z 207.577,A -85,B 0,C 180,E1 -17910,E2 -17910} C_VEL
LIN {X 0,Y 381.313,Z 207.518,A -85,B 0,C 180,E1 -17911.584,E2 -17911.584} C_VEL
LIN {X 0,Y 380.222,Z 206.976,A -85,B 0,C 180,E1 -17913.513,E2 -17913.513} C_VEL
LIN {X 0,Y 378.214,Z 206.267,A -85,B 0,C 180,E1 -17915.49,E2 -17915.49} C_VEL
LIN {X 0,Y 375.564,Z 204.905,A -85,B 0,C 180,E1 -17917.348,E2 -17917.348} C_VEL
LIN {X 0,Y 372.203,Z 202.799,A -85,B 0,C 180,E1 -17919.177,E2 -17919.177} C_VEL
LIN {X 0,Y 368.461,Z 199.872,A -85,B 0,C 180,E1 -17920.883,E2 -17920.883} C_VEL
LIN {X 0,Y 366.019,Z 197.979,A -85,B 0,C 180,E1 -17921.856,E2 -17921.856} C_VEL
LIN {X 0,Y 361.119,Z 195.047,A -85,B 0,C 180,E1 -17923.559,E2 -17923.559} C_VEL
LIN {X 0,Y 355.434,Z 190.699,A -85,B 0,C 180,E1 -17925.317,E2 -17925.317} C_VEL
LIN {X 0,Y 348.215,Z 185.43,A -85,B 0,C 180,E1 -17927.249,E2 -17927.249} C_VEL
LIN {X 0,Y 342.62,Z 180.682,A -85,B 0,C 180,E1 -17928.623,E2 -17928.623} C_VEL
LIN {X 0,Y 335.814,Z 175.497,A -85,B 0,C 180,E1 -17930.124,E2 -17930.124} C_VEL
LIN {X 0,Y 327.645,Z 168.514,A -85,B 0,C 180,E1 -17931.774,E2 -17931.774} C_VEL
LIN {X 0,Y 318.765,Z 160.448,A -85,B 0,C 180,E1 -17933.356,E2 -17933.356} C_VEL
LIN {X 0,Y 309.767,Z 151.971,A -85,B 0,C 180,E1 -17934.728,E2 -17934.728} C_VEL
LIN {X 0,Y 301.2,Z 143.246,A -85,B 0,C 180,E1 -17935.858,E2 -17935.858} C_VEL
LIN {X 0,Y 290.619,Z 131.43,A -85,B 0,C 180,E1 -17937.206,E2 -17937.206} C_VEL
LIN {X 0,Y 282.327,Z 119.525,A -85,B 0,C 180,E1 -17938.419,E2 -17938.419} C_VEL
LIN {X 0,Y 271.295,Z 99.282,A -85,B 0,C 180,E1 -17940.305,E2 -17940.305} C_VEL
LIN {X 0,Y 270.369,Z 97.017,A -85,B 0,C 180,E1 -17940.563,E2 -17940.563} C_VEL
LIN {X 0,Y 270.204,Z 96.375,A -85,B 0,C 180,E1 -17940.872,E2 -17940.872} C_VEL
LIN {X 0,Y 270.211,Z 96.288,A -85,B 0,C 180,E1 -17944.904,E2 -17944.904} C_VEL
LIN {X 0,Y 270.219,Z 96.32,A -85,B 0,C 180,E1 -17948.717,E2 -17948.717} C_VEL
LIN {X 0,Y 270.161,Z 96.281,A -85,B 0,C 180,E1 -17953.249,E2 -17953.249} C_VEL
LIN {X 0,Y 270.181,Z 96.327,A -85,B 0,C 180,E1 -17957.445,E2 -17957.445} C_VEL
LIN {X 0,Y 270.242,Z 96.32,A -85,B 0,C 180,E1 -17961.381,E2 -17961.381} C_VEL
LIN {X 0,Y 270.213,Z 96.304,A -85,B 0,C 180,E1 -17965.097,E2 -17965.097} C_VEL
LIN {X 0,Y 270.198,Z 96.33,A -85,B 0,C 180,E1 -17969.131,E2 -17969.131} C_VEL
LIN {X 0,Y 270.261,Z 96.292,A -85,B 0,C 180,E1 -17972.147,E2 -17972.147} C_VEL
LIN {X 0,Y 270.275,Z 96.315,A -85,B 0,C 180,E1 -17975.52,E2 -17975.52} C_VEL
LIN {X 0,Y 270.3,Z 96.282,A -85,B 0,C 180,E1 -17980.245,E2 -17980.245} C_VEL
LIN {X 0,Y 270.402,Z 96.304,A -85,B 0,C 180,E1 -17984.936,E2 -17984.936} C_VEL
LIN {X 0,Y 270.442,Z 96.259,A -85,B 0,C 180,E1 -17989.52,E2 -17989.52} C_VEL
LIN {X 0,Y 270.611,Z 96.258,A -85,B 0,C 180,E1 -17992.54,E2 -17992.54} C_VEL
LIN {X 0,Y 270.786,Z 96.222,A -85,B 0,C 180,E1 -17998.514,E2 -17998.514} C_VEL
LIN {X 0,Y 270.786,Z 96.225,A -85,B 0,C 180,E1 -18001.488,E2 -18001.488} C_VEL
LIN {X 0,Y 270.613,Z 96.255,A -85,B 0,C 180,E1 -18007.462,E2 -18007.462} C_VEL
LIN {X 0,Y 270.442,Z 96.258,A -85,B 0,C 180,E1 -18010.482,E2 -18010.482} C_VEL
LIN {X 0,Y 270.404,Z 96.3,A -85,B 0,C 180,E1 -18015.065,E2 -18015.065} C_VEL
LIN {X 0,Y 270.303,Z 96.28,A -85,B 0,C 180,E1 -18019.756,E2 -18019.756} C_VEL
LIN {X 0,Y 270.275,Z 96.309,A -85,B 0,C 180,E1 -18024.586,E2 -18024.586} C_VEL
LIN {X 0,Y 270.271,Z 96.292,A -85,B 0,C 180,E1 -18027.909,E2 -18027.909} C_VEL
LIN {X 0,Y 270.186,Z 96.328,A -85,B 0,C 180,E1 -18031.349,E2 -18031.349} C_VEL
LIN {X 0,Y 270.18,Z 96.312,A -85,B 0,C 180,E1 -18032.749,E2 -18032.749} C_VEL
LIN {X 0,Y 269.566,Z 96.388,A -85,B 0,C 180,E1 -18033.994,E2 -18033.994} C_VEL
LIN {X 0,Y 266.731,Z 96.751,A -85,B 0,C 180,E1 -18036.023,E2 -18036.023} C_VEL
LIN {X 0,Y 264.28,Z 97.065,A -85,B 0,C 180,E1 -18037.672,E2 -18037.672} C_VEL
LIN {X 0,Y 263.209,Z 97.188,A -85,B 0,C 180,E1 -18038.951,E2 -18038.951} C_VEL
LIN {X 0,Y 263.114,Z 97.196,A -85,B 0,C 180,E1 -18039.384,E2 -18039.384} C_VEL
LIN {X 0,Y 263.126,Z 97.207,A -85,B 0,C 180,E1 -18041.894,E2 -18041.894} C_VEL
LIN {X 0,Y 263.126,Z 97.207,A -85,B 0,C 180,E1 -18046.151,E2 -18046.151} C_VEL
LIN {X 0,Y 263.117,Z 97.176,A -85,B 0,C 180,E1 -18050.13,E2 -18050.13} C_VEL
LIN {X 0,Y 263.228,Z 97.365,A -85,B 0,C 180,E1 -18051.698,E2 -18051.698} C_VEL
LIN {X 0,Y 264.78,Z 104.536,A -85,B 0,C 180,E1 -18055.37,E2 -18055.37} C_VEL
LIN {X 0,Y 266.283,Z 112.179,A -85,B 0,C 180,E1 -18059.005,E2 -18059.005} C_VEL
LIN {X 0,Y 268.242,Z 116.938,A -85,B 0,C 180,E1 -18059.471,E2 -18059.471} C_VEL
LIN {X 0,Y 272.497,Z 127.185,A -85,B 0,C 180,E1 -18060.298,E2 -18060.298} C_VEL
LIN {X 0,Y 277.245,Z 150.212,A -85,B 0,C 180,E1 -18061.517,E2 -18061.517} C_VEL
LIN {X 0,Y 279.174,Z 162.628,A -85,B 0,C 180,E1 -18062.084,E2 -18062.084} C_VEL
LIN {X 0,Y 277.46,Z 218.362,A -85,B 0,C 180,E1 -18063.535,E2 -18063.535} C_VEL
LIN {X 0,Y 276.699,Z 228.651,A -85,B 0,C 180,E1 -18063.964,E2 -18063.964} C_VEL
LIN {X 0,Y 275.696,Z 238.162,A -85,B 0,C 180,E1 -18064.521,E2 -18064.521} C_VEL
LIN {X 0,Y 274.575,Z 247.235,A -85,B 0,C 180,E1 -18065.22,E2 -18065.22} C_VEL
LIN {X 0,Y 273.204,Z 256.365,A -85,B 0,C 180,E1 -18066.099,E2 -18066.099} C_VEL
LIN {X 0,Y 271.678,Z 265.358,A -85,B 0,C 180,E1 -18067.168,E2 -18067.168} C_VEL
LIN {X 0,Y 270.06,Z 274.084,A -85,B 0,C 180,E1 -18068.433,E2 -18068.433} C_VEL
LIN {X 0,Y 268.581,Z 281.476,A -85,B 0,C 180,E1 -18069.714,E2 -18069.714} C_VEL
LIN {X 0,Y 267.055,Z 288.858,A -85,B 0,C 180,E1 -18071.233,E2 -18071.233} C_VEL
LIN {X 0,Y 265.879,Z 294.953,A -85,B 0,C 180,E1 -18072.716,E2 -18072.716} C_VEL
LIN {X 0,Y 264.506,Z 301.435,A -85,B 0,C 180,E1 -18074.591,E2 -18074.591} C_VEL
LIN {X 0,Y 263.504,Z 305.935,A -85,B 0,C 180,E1 -18076.111,E2 -18076.111} C_VEL
LIN {X 0,Y 262.389,Z 311.428,A -85,B 0,C 180,E1 -18078.411,E2 -18078.411} C_VEL
LIN {X 0,Y 261.686,Z 315.756,A -85,B 0,C 180,E1 -18080.727,E2 -18080.727} C_VEL
LIN {X 0,Y 261.353,Z 318.124,A -85,B 0,C 180,E1 -18082.273,E2 -18082.273} C_VEL
LIN {X 0,Y 261.056,Z 320.988,A -85,B 0,C 180,E1 -18084.941,E2 -18084.941} C_VEL
LIN {X 0,Y 261.052,Z 322.378,A -85,B 0,C 180,E1 -18086.914,E2 -18086.914} C_VEL
LIN {X 0,Y 261.088,Z 322.97,A -85,B 0,C 180,E1 -18088.458,E2 -18088.458} C_VEL
LIN {X 0,Y 261.127,Z 323.125,A -85,B 0,C 180,E1 -18090,E2 -18090} C_VEL
LIN {X 0,Y 261.088,Z 322.97,A -85,B 0,C 180,E1 -18091.542,E2 -18091.542} C_VEL
LIN {X 0,Y 261.052,Z 322.378,A -85,B 0,C 180,E1 -18093.086,E2 -18093.086} C_VEL
LIN {X 0,Y 261.153,Z 319.926,A -85,B 0,C 180,E1 -18096.18,E2 -18096.18} C_VEL
LIN {X 0,Y 261.51,Z 316.974,A -85,B 0,C 180,E1 -18098.5,E2 -18098.5} C_VEL
LIN {X 0,Y 262.114,Z 312.982,A -85,B 0,C 180,E1 -18100.818,E2 -18100.818} C_VEL
LIN {X 0,Y 263.07,Z 307.851,A -85,B 0,C 180,E1 -18103.125,E2 -18103.125} C_VEL
LIN {X 0,Y 264.234,Z 302.59,A -85,B 0,C 180,E1 -18105.03,E2 -18105.03} C_VEL
LIN {X 0,Y 265.568,Z 296.273,A -85,B 0,C 180,E1 -18106.924,E2 -18106.924} C_VEL
LIN {X 0,Y 266.867,Z 290.324,A -85,B 0,C 180,E1 -18108.423,E2 -18108.423} C_VEL
LIN {X 0,Y 268.22,Z 283.396,A -85,B 0,C 180,E1 -18109.915,E2 -18109.915} C_VEL
LIN {X 0,Y 269.858,Z 275.219,A -85,B 0,C 180,E1 -18111.383,E2 -18111.383} C_VEL
LIN {X 0,Y 271.456,Z 266.71,A -85,B 0,C 180,E1 -18112.651,E2 -18112.651} C_VEL
LIN {X 0,Y 272.969,Z 257.998,A -85,B 0,C 180,E1 -18113.721,E2 -18113.721} C_VEL
LIN {X 0,Y 274.411,Z 248.241,A -85,B 0,C 180,E1 -18114.695,E2 -18114.695} C_VEL
LIN {X 0,Y 275.528,Z 239.449,A -85,B 0,C 180,E1 -18115.394,E2 -18115.394} C_VEL
LIN {X 0,Y 276.597,Z 229.524,A -85,B 0,C 180,E1 -18115.996,E2 -18115.996} C_VEL
LIN {X 0,Y 277.318,Z 219.669,A -85,B 0,C 180,E1 -18116.429,E2 -18116.429} C_VEL
LIN {X 0,Y 278.123,Z 196.846,A -85,B 0,C 180,E1 -18117.055,E2 -18117.055} C_VEL
LIN {X 0,Y 279.121,Z 161.724,A -85,B 0,C 180,E1 -18117.947,E2 -18117.947} C_VEL
LIN {X 0,Y 275.75,Z 142.446,A -85,B 0,C 180,E1 -18118.876,E2 -18118.876} C_VEL
LIN {X 0,Y 272.204,Z 126.203,A -85,B 0,C 180,E1 -18119.766,E2 -18119.766} C_VEL
LIN {X 0,Y 266.381,Z 112.533,A -85,B 0,C 180,E1 -18120.931,E2 -18120.931} C_VEL
LIN {X 0,Y 266.106,Z 111.345,A -85,B 0,C 180,E1 -18121.296,E2 -18121.296} C_VEL
LIN {X 0,Y 264.589,Z 103.597,A -85,B 0,C 180,E1 -18125.095,E2 -18125.095} C_VEL
LIN {X 0,Y 263.217,Z 97.287,A -85,B 0,C 180,E1 -18128.364,E2 -18128.364} C_VEL
LIN {X 0,Y 263.126,Z 97.19,A -85,B 0,C 180,E1 -18131.893,E2 -18131.893} C_VEL
LIN {X 0,Y 263.107,Z 97.205,A -85,B 0,C 180,E1 -18136.154,E2 -18136.154} C_VEL
LIN {X 0,Y 263.107,Z 97.195,A -85,B 0,C 180,E1 -18140.127,E2 -18140.127} C_VEL
LIN {X 0,Y 263.165,Z 97.194,A -85,B 0,C 180,E1 -18144.018,E2 -18144.018} C_VEL
LIN {X 0,Y 263.134,Z 97.199,A -85,B 0,C 180,E1 -18147.711,E2 -18147.711} C_VEL
LIN {X 0,Y 263.197,Z 97.176,A -85,B 0,C 180,E1 -18151.785,E2 -18151.785} C_VEL
LIN {X 0,Y 263.227,Z 97.183,A -85,B 0,C 180,E1 -18155.2,E2 -18155.2} C_VEL
LIN {X 0,Y 263.265,Z 97.163,A -85,B 0,C 180,E1 -18159.693,E2 -18159.693} C_VEL
LIN {X 0,Y 263.352,Z 97.173,A -85,B 0,C 180,E1 -18164.521,E2 -18164.521} C_VEL
LIN {X 0,Y 263.375,Z 97.14,A -85,B 0,C 180,E1 -18169.234,E2 -18169.234} C_VEL
LIN {X 0,Y 263.574,Z 97.129,A -85,B 0,C 180,E1 -18172.338,E2 -18172.338} C_VEL
LIN {X 0,Y 263.751,Z 97.101,A -85,B 0,C 180,E1 -18178.472,E2 -18178.472} C_VEL
LIN {X 0,Y 263.751,Z 97.098,A -85,B 0,C 180,E1 -18181.526,E2 -18181.526} C_VEL
LIN {X 0,Y 263.572,Z 97.132,A -85,B 0,C 180,E1 -18187.661,E2 -18187.661} C_VEL
LIN {X 0,Y 263.374,Z 97.141,A -85,B 0,C 180,E1 -18190.765,E2 -18190.765} C_VEL
LIN {X 0,Y 263.35,Z 97.178,A -85,B 0,C 180,E1 -18195.477,E2 -18195.477} C_VEL
LIN {X 0,Y 263.262,Z 97.163,A -85,B 0,C 180,E1 -18200.306,E2 -18200.306} C_VEL
LIN {X 0,Y 263.206,Z 97.185,A -85,B 0,C 180,E1 -18205.291,E2 -18205.291} C_VEL
LIN {X 0,Y 263.163,Z 97.185,A -85,B 0,C 180,E1 -18208.73,E2 -18208.73} C_VEL
LIN {X 0,Y 263.131,Z 97.203,A -85,B 0,C 180,E1 -18212.287,E2 -18212.287} C_VEL
LIN {X 0,Y 263.186,Z 97.189,A -85,B 0,C 180,E1 -18215.977,E2 -18215.977} C_VEL
LIN {X 0,Y 263.135,Z 97.192,A -85,B 0,C 180,E1 -18219.866,E2 -18219.866} C_VEL
LIN {X 0,Y 263.124,Z 97.207,A -85,B 0,C 180,E1 -18223.983,E2 -18223.983} C_VEL
LIN {X 0,Y 263.121,Z 97.151,A -85,B 0,C 180,E1 -18228.406,E2 -18228.406} C_VEL
LIN {X 0,Y 263.162,Z 97.208,A -85,B 0,C 180,E1 -18232.104,E2 -18232.104} C_VEL
LIN {X 0,Y 263.18,Z 97.165,A -85,B 0,C 180,E1 -18235.89,E2 -18235.89} C_VEL
LIN {X 0,Y 263.17,Z 97.409,A -85,B 0,C 180,E1 -18238.398,E2 -18238.398} C_VEL
LIN {X 0,Y 263.397,Z 98.378,A -85,B 0,C 180,E1 -18238.629,E2 -18238.629} C_VEL
LIN {X 0,Y 271.858,Z 114.16,A -85,B 0,C 180,E1 -18240.211,E2 -18240.211} C_VEL
LIN {X 0,Y 278.524,Z 125.929,A -85,B 0,C 180,E1 -18241.338,E2 -18241.338} C_VEL
LIN {X 0,Y 286.764,Z 137.474,A -85,B 0,C 180,E1 -18242.562,E2 -18242.562} C_VEL
LIN {X 0,Y 297.132,Z 149.021,A -85,B 0,C 180,E1 -18243.909,E2 -18243.909} C_VEL
LIN {X 0,Y 308.023,Z 159.738,A -85,B 0,C 180,E1 -18245.281,E2 -18245.281} C_VEL
LIN {X 0,Y 316.751,Z 167.722,A -85,B 0,C 180,E1 -18246.576,E2 -18246.576} C_VEL
LIN {X 0,Y 324.789,Z 174.866,A -85,B 0,C 180,E1 -18247.958,E2 -18247.958} C_VEL
LIN {X 0,Y 332.294,Z 181.123,A -85,B 0,C 180,E1 -18249.407,E2 -18249.407} C_VEL
LIN {X 0,Y 339.013,Z 186.308,A -85,B 0,C 180,E1 -18250.832,E2 -18250.832} C_VEL
LIN {X 0,Y 346.471,Z 192.327,A -85,B 0,C 180,E1 -18252.589,E2 -18252.589} C_VEL
LIN {X 0,Y 352.782,Z 196.844,A -85,B 0,C 180,E1 -18254.248,E2 -18254.248} C_VEL
LIN {X 0,Y 358.008,Z 200.864,A -85,B 0,C 180,E1 -18255.788,E2 -18255.788} C_VEL
LIN {X 0,Y 362.863,Z 203.897,A -85,B 0,C 180,E1 -18257.36,E2 -18257.36} C_VEL
LIN {X 0,Y 366.201,Z 205.97,A -85,B 0,C 180,E1 -18258.579,E2 -18258.579} C_VEL
LIN {X 0,Y 370.18,Z 209.161,A -85,B 0,C 180,E1 -18260.299,E2 -18260.299} C_VEL
LIN {X 0,Y 373.567,Z 211.363,A -85,B 0,C 180,E1 -18262.024,E2 -18262.024} C_VEL
LIN {X 0,Y 376.501,Z 212.946,A -85,B 0,C 180,E1 -18263.884,E2 -18263.884} C_VEL
LIN {X 0,Y 378.681,Z 213.846,A -85,B 0,C 180,E1 -18265.743,E2 -18265.743} C_VEL
LIN {X 0,Y 379.929,Z 214.267,A -85,B 0,C 180,E1 -18267.3,E2 -18267.3} C_VEL
LIN {X 0,Y 380.607,Z 214.738,A -85,B 0,C 180,E1 -18268.942,E2 -18268.942} C_VEL
LIN {X 0,Y 380.758,Z 214.623,A -85,B 0,C 180,E1 -18270,E2 -18270} C_VEL
LIN {X 0,Y 380.444,Z 214.565,A -85,B 0,C 180,E1 -18271.588,E2 -18271.588} C_VEL
LIN {X 0,Y 379.6,Z 214.062,A -85,B 0,C 180,E1 -18273.184,E2 -18273.184} C_VEL
LIN {X 0,Y 377.821,Z 213.524,A -85,B 0,C 180,E1 -18275.065,E2 -18275.065} C_VEL
LIN {X 0,Y 375.25,Z 212.305,A -85,B 0,C 180,E1 -18276.967,E2 -18276.967} C_VEL
LIN {X 0,Y 371.894,Z 210.314,A -85,B 0,C 180,E1 -18278.873,E2 -18278.873} C_VEL
LIN {X 0,Y 368.047,Z 207.566,A -85,B 0,C 180,E1 -18280.654,E2 -18280.654} C_VEL
LIN {X 0,Y 364.633,Z 204.869,A -85,B 0,C 180,E1 -18282.014,E2 -18282.014} C_VEL
LIN {X 0,Y 359.521,Z 201.86,A -85,B 0,C 180,E1 -18283.754,E2 -18283.754} C_VEL
LIN {X 0,Y 353.673,Z 197.563,A -85,B 0,C 180,E1 -18285.504,E2 -18285.504} C_VEL
LIN {X 0,Y 348.807,Z 193.964,A -85,B 0,C 180,E1 -18286.817,E2 -18286.817} C_VEL
LIN {X 0,Y 342.384,Z 189.153,A -85,B 0,C 180,E1 -18288.391,E2 -18288.391} C_VEL
LIN {X 0,Y 337.563,Z 185.228,A -85,B 0,C 180,E1 -18289.487,E2 -18289.487} C_VEL
LIN {X 0,Y 331.399,Z 180.351,A -85,B 0,C 180,E1 -18290.776,E2 -18290.776} C_VEL
LIN {X 0,Y 323.554,Z 173.833,A -85,B 0,C 180,E1 -18292.252,E2 -18292.252} C_VEL
LIN {X 0,Y 316.116,Z 167.14,A -85,B 0,C 180,E1 -18293.531,E2 -18293.531} C_VEL
LIN {X 0,Y 306.56,Z 158.426,A -85,B 0,C 180,E1 -18294.91,E2 -18294.91} C_VEL
LIN {X 0,Y 296.081,Z 147.846,A -85,B 0,C 180,E1 -18296.223,E2 -18296.223} C_VEL
LIN {X 0,Y 286.115,Z 136.685,A -85,B 0,C 180,E1 -18297.528,E2 -18297.528} C_VEL
LIN {X 0,Y 278.047,Z 125.177,A -85,B 0,C 180,E1 -18298.737,E2 -18298.737} C_VEL
LIN {X 0,Y 271.756,Z 113.972,A -85,B 0,C 180,E1 -18299.807,E2 -18299.807} C_VEL
LIN {X 0,Y 264.619,Z 100.734,A -85,B 0,C 180,E1 -18301.115,E2 -18301.115} C_VEL
LIN {X 0,Y 263.301,Z 98.042,A -85,B 0,C 180,E1 -18301.428,E2 -18301.428} C_VEL
LIN {X 0,Y 263.126,Z 97.264,A -85,B 0,C 180,E1 -18301.787,E2 -18301.787} C_VEL
LIN {X 0,Y 263.17,Z 97.166,A -85,B 0,C 180,E1 -18304.122,E2 -18304.122} C_VEL
LIN {X 0,Y 263.162,Z 97.208,A -85,B 0,C 180,E1 -18307.896,E2 -18307.896} C_VEL
LIN {X 0,Y 263.12,Z 97.15,A -85,B 0,C 180,E1 -18311.894,E2 -18311.894} C_VEL
LIN {X 0,Y 263.126,Z 97.209,A -85,B 0,C 180,E1 -18316.15,E2 -18316.15} C_VEL
LIN {X 0,Y 263.135,Z 97.192,A -85,B 0,C 180,E1 -18320.134,E2 -18320.134} C_VEL
LIN {X 0,Y 263.186,Z 97.189,A -85,B 0,C 180,E1 -18324.023,E2 -18324.023} C_VEL
LIN {X 0,Y 263.131,Z 97.203,A -85,B 0,C 180,E1 -18327.713,E2 -18327.713} C_VEL
LIN {X 0,Y 263.194,Z 97.175,A -85,B 0,C 180,E1 -18331.786,E2 -18331.786} C_VEL
LIN {X 0,Y 263.224,Z 97.188,A -85,B 0,C 180,E1 -18335.201,E2 -18335.201} C_VEL
LIN {X 0,Y 263.262,Z 97.163,A -85,B 0,C 180,E1 -18339.694,E2 -18339.694} C_VEL
LIN {X 0,Y 263.35,Z 97.178,A -85,B 0,C 180,E1 -18344.523,E2 -18344.523} C_VEL
LIN {X 0,Y 263.374,Z 97.141,A -85,B 0,C 180,E1 -18349.235,E2 -18349.235} C_VEL
LIN {X 0,Y 263.572,Z 97.132,A -85,B 0,C 180,E1 -18352.339,E2 -18352.339} C_VEL
LIN {X 0,Y 263.751,Z 97.098,A -85,B 0,C 180,E1 -18358.474,E2 -18358.474} C_VEL
LIN {X 0,Y 263.751,Z 97.101,A -85,B 0,C 180,E1 -18361.528,E2 -18361.528} C_VEL
LIN {X 0,Y 263.574,Z 97.129,A -85,B 0,C 180,E1 -18367.662,E2 -18367.662} C_VEL
LIN {X 0,Y 263.375,Z 97.14,A -85,B 0,C 180,E1 -18370.766,E2 -18370.766} C_VEL
LIN {X 0,Y 263.352,Z 97.173,A -85,B 0,C 180,E1 -18375.479,E2 -18375.479} C_VEL
LIN {X 0,Y 263.265,Z 97.163,A -85,B 0,C 180,E1 -18380.307,E2 -18380.307} C_VEL
LIN {X 0,Y 263.21,Z 97.18,A -85,B 0,C 180,E1 -18385.292,E2 -18385.292} C_VEL
LIN {X 0,Y 263.167,Z 97.187,A -85,B 0,C 180,E1 -18388.732,E2 -18388.732} C_VEL
LIN {X 0,Y 263.114,Z 97.194,A -85,B 0,C 180,E1 -18392.741,E2 -18392.741} C_VEL
LIN {X 0,Y 263.185,Z 97.199,A -85,B 0,C 180,E1 -18396.764,E2 -18396.764} C_VEL
LIN {X 0,Y 263.114,Z 97.196,A -85,B 0,C 180,E1 -18399.384,E2 -18399.384} C_VEL
LIN {X 0,Y 262.417,Z 97.284,A -85,B 0,C 180,E1 -18400.662,E2 -18400.662} C_VEL
LIN {X 0,Y 259.539,Z 97.658,A -85,B 0,C 180,E1 -18402.744,E2 -18402.744} C_VEL
LIN {X 0,Y 257.126,Z 97.951,A -85,B 0,C 180,E1 -18404.438,E2 -18404.438} C_VEL
LIN {X 0,Y 256.114,Z 98.075,A -85,B 0,C 180,E1 -18405.751,E2 -18405.751} C_VEL
LIN {X 0,Y 256.043,Z 98.087,A -85,B 0,C 180,E1 -18406.196,E2 -18406.196} C_VEL
LIN {X 0,Y 256.095,Z 98.064,A -85,B 0,C 180,E1 -18410.703,E2 -18410.703} C_VEL
LIN {X 0,Y 256.291,Z 98.837,A -85,B 0,C 180,E1 -18411.346,E2 -18411.346} C_VEL
LIN {X 0,Y 257.477,Z 103.958,A -85,B 0,C 180,E1 -18414.067,E2 -18414.067} C_VEL
LIN {X 0,Y 259.015,Z 111.814,A -85,B 0,C 180,E1 -18417.994,E2 -18417.994} C_VEL
LIN {X 0,Y 259.795,Z 114.19,A -85,B 0,C 180,E1 -18418.287,E2 -18418.287} C_VEL
LIN {X 0,Y 265.698,Z 127.381,A -85,B 0,C 180,E1 -18419.47,E2 -18419.47} C_VEL
LIN {X 0,Y 267.125,Z 131.891,A -85,B 0,C 180,E1 -18419.787,E2 -18419.787} C_VEL
LIN {X 0,Y 271.448,Z 154.111,A -85,B 0,C 180,E1 -18420.972,E2 -18420.972} C_VEL
LIN {X 0,Y 272.867,Z 163.5,A -85,B 0,C 180,E1 -18421.411,E2 -18421.411} C_VEL
LIN {X 0,Y 271.119,Z 218.361,A -85,B 0,C 180,E1 -18422.874,E2 -18422.874} C_VEL
LIN {X 0,Y 270.249,Z 229.387,A -85,B 0,C 180,E1 -18423.35,E2 -18423.35} C_VEL
LIN {X 0,Y 268.849,Z 241.832,A -85,B 0,C 180,E1 -18424.137,E2 -18424.137} C_VEL
LIN {X 0,Y 267.019,Z 254.544,A -85,B 0,C 180,E1 -18425.302,E2 -18425.302} C_VEL
LIN {X 0,Y 265.405,Z 263.817,A -85,B 0,C 180,E1 -18426.39,E2 -18426.39} C_VEL
LIN {X 0,Y 263.696,Z 272.759,A -85,B 0,C 180,E1 -18427.679,E2 -18427.679} C_VEL
LIN {X 0,Y 261.929,Z 281.286,A -85,B 0,C 180,E1 -18429.175,E2 -18429.175} C_VEL
LIN {X 0,Y 260.353,Z 288.503,A -85,B 0,C 180,E1 -18430.69,E2 -18430.69} C_VEL
LIN {X 0,Y 258.761,Z 296.082,A -85,B 0,C 180,E1 -18432.617,E2 -18432.617} C_VEL
LIN {X 0,Y 257.362,Z 302.399,A -85,B 0,C 180,E1 -18434.559,E2 -18434.559} C_VEL
LIN {X 0,Y 256.122,Z 307.659,A -85,B 0,C 180,E1 -18436.512,E2 -18436.512} C_VEL
LIN {X 0,Y 255.106,Z 312.791,A -85,B 0,C 180,E1 -18438.881,E2 -18438.881} C_VEL
LIN {X 0,Y 254.466,Z 316.782,A -85,B 0,C 180,E1 -18441.263,E2 -18441.263} C_VEL
LIN {X 0,Y 254.066,Z 319.735,A -85,B 0,C 180,E1 -18443.647,E2 -18443.647} C_VEL
LIN {X 0,Y 253.952,Z 322.187,A -85,B 0,C 180,E1 -18446.827,E2 -18446.827} C_VEL
LIN {X 0,Y 253.995,Z 322.779,A -85,B 0,C 180,E1 -18448.414,E2 -18448.414} C_VEL
LIN {X 0,Y 254.055,Z 322.936,A -85,B 0,C 180,E1 -18450,E2 -18450} C_VEL
LIN {X 0,Y 253.995,Z 322.779,A -85,B 0,C 180,E1 -18451.586,E2 -18451.586} C_VEL
LIN {X 0,Y 253.951,Z 322.187,A -85,B 0,C 180,E1 -18453.173,E2 -18453.173} C_VEL
LIN {X 0,Y 254.066,Z 319.735,A -85,B 0,C 180,E1 -18456.353,E2 -18456.353} C_VEL
LIN {X 0,Y 254.466,Z 316.782,A -85,B 0,C 180,E1 -18458.737,E2 -18458.737} C_VEL
LIN {X 0,Y 255.106,Z 312.791,A -85,B 0,C 180,E1 -18461.119,E2 -18461.119} C_VEL
LIN {X 0,Y 256.12,Z 307.659,A -85,B 0,C 180,E1 -18463.488,E2 -18463.488} C_VEL
LIN {X 0,Y 257.365,Z 302.399,A -85,B 0,C 180,E1 -18465.441,E2 -18465.441} C_VEL
LIN {X 0,Y 258.777,Z 296.083,A -85,B 0,C 180,E1 -18467.382,E2 -18467.382} C_VEL
LIN {X 0,Y 260.154,Z 289.803,A -85,B 0,C 180,E1 -18468.998,E2 -18468.998} C_VEL
LIN {X 0,Y 261.52,Z 283.204,A -85,B 0,C 180,E1 -18470.448,E2 -18470.448} C_VEL
LIN {X 0,Y 263.233,Z 275.028,A -85,B 0,C 180,E1 -18471.949,E2 -18471.949} C_VEL
LIN {X 0,Y 264.909,Z 266.519,A -85,B 0,C 180,E1 -18473.243,E2 -18473.243} C_VEL
LIN {X 0,Y 266.484,Z 257.807,A -85,B 0,C 180,E1 -18474.335,E2 -18474.335} C_VEL
LIN {X 0,Y 267.981,Z 248.051,A -85,B 0,C 180,E1 -18475.328,E2 -18475.328} C_VEL
LIN {X 0,Y 269.332,Z 237.973,A -85,B 0,C 180,E1 -18476.125,E2 -18476.125} C_VEL
LIN {X 0,Y 270.3,Z 228.525,A -85,B 0,C 180,E1 -18476.696,E2 -18476.696} C_VEL
LIN {X 0,Y 271.05,Z 218.359,A -85,B 0,C 180,E1 -18477.133,E2 -18477.133} C_VEL
LIN {X 0,Y 272.859,Z 164.834,A -85,B 0,C 180,E1 -18478.55,E2 -18478.55} C_VEL
LIN {X 0,Y 272.624,Z 161.287,A -85,B 0,C 180,E1 -18478.681,E2 -18478.681} C_VEL
LIN {X 0,Y 268.911,Z 140.547,A -85,B 0,C 180,E1 -18479.733,E2 -18479.733} C_VEL
LIN {X 0,Y 266.346,Z 128.984,A -85,B 0,C 180,E1 -18480.399,E2 -18480.399} C_VEL
LIN {X 0,Y 260.188,Z 114.934,A -85,B 0,C 180,E1 -18481.636,E2 -18481.636} C_VEL
LIN {X 0,Y 259.076,Z 111.971,A -85,B 0,C 180,E1 -18481.954,E2 -18481.954} C_VEL
LIN {X 0,Y 257.768,Z 105.536,A -85,B 0,C 180,E1 -18485.119,E2 -18485.119} C_VEL
LIN {X 0,Y 256.291,Z 98.839,A -85,B 0,C 180,E1 -18488.653,E2 -18488.653} C_VEL
LIN {X 0,Y 256.095,Z 98.066,A -85,B 0,C 180,E1 -18489.297,E2 -18489.297} C_VEL
LIN {X 0,Y 256.064,Z 98.092,A -85,B 0,C 180,E1 -18493.326,E2 -18493.326} C_VEL
LIN {X 0,Y 256.072,Z 98.088,A -85,B 0,C 180,E1 -18497.819,E2 -18497.819} C_VEL
LIN {X 0,Y 256.073,Z 98.075,A -85,B 0,C 180,E1 -18500.857,E2 -18500.857} C_VEL
LIN {X 0,Y 256.133,Z 98.081,A -85,B 0,C 180,E1 -18502.867,E2 -18502.867} C_VEL
LIN {X 0,Y 256.069,Z 98.066,A -85,B 0,C 180,E1 -18506.707,E2 -18506.707} C_VEL
LIN {X 0,Y 256.105,Z 98.077,A -85,B 0,C 180,E1 -18510.398,E2 -18510.398} C_VEL
LIN {X 0,Y 256.19,Z 98.055,A -85,B 0,C 180,E1 -18514.861,E2 -18514.861} C_VEL
LIN {X 0,Y 256.168,Z 98.056,A -85,B 0,C 180,E1 -18519.104,E2 -18519.104} C_VEL
LIN {X 0,Y 256.301,Z 98.048,A -85,B 0,C 180,E1 -18524.084,E2 -18524.084} C_VEL
LIN {X 0,Y 256.311,Z 98.023,A -85,B 0,C 180,E1 -18528.933,E2 -18528.933} C_VEL
LIN {X 0,Y 256.541,Z 98.002,A -85,B 0,C 180,E1 -18532.126,E2 -18532.126} C_VEL
LIN {X 0,Y 256.714,Z 97.977,A -85,B 0,C 180,E1 -18538.43,E2 -18538.43} C_VEL
LIN {X 0,Y 256.714,Z 97.974,A -85,B 0,C 180,E1 -18541.568,E2 -18541.568} C_VEL
LIN {X 0,Y 256.54,Z 98.005,A -85,B 0,C 180,E1 -18547.872,E2 -18547.872} C_VEL
LIN {X 0,Y 256.31,Z 98.023,A -85,B 0,C 180,E1 -18551.065,E2 -18551.065} C_VEL
LIN {X 0,Y 256.299,Z 98.053,A -85,B 0,C 180,E1 -18555.914,E2 -18555.914} C_VEL
LIN {X 0,Y 256.165,Z 98.055,A -85,B 0,C 180,E1 -18560.894,E2 -18560.894} C_VEL
LIN {X 0,Y 256.187,Z 98.061,A -85,B 0,C 180,E1 -18565.138,E2 -18565.138} C_VEL
LIN {X 0,Y 256.101,Z 98.075,A -85,B 0,C 180,E1 -18569.6,E2 -18569.6} C_VEL
LIN {X 0,Y 256.083,Z 98.069,A -85,B 0,C 180,E1 -18573.289,E2 -18573.289} C_VEL
LIN {X 0,Y 256.138,Z 98.082,A -85,B 0,C 180,E1 -18577.278,E2 -18577.278} C_VEL
LIN {X 0,Y 256.07,Z 98.07,A -85,B 0,C 180,E1 -18581.199,E2 -18581.199} C_VEL
LIN {X 0,Y 256.042,Z 98.058,A -85,B 0,C 180,E1 -18585.532,E2 -18585.532} C_VEL
LIN {X 0,Y 256.052,Z 98.032,A -85,B 0,C 180,E1 -18588.796,E2 -18588.796} C_VEL
LIN {X 0,Y 256.142,Z 98.069,A -85,B 0,C 180,E1 -18592.869,E2 -18592.869} C_VEL
LIN {X 0,Y 256.097,Z 98.11,A -85,B 0,C 180,E1 -18597.302,E2 -18597.302} C_VEL
LIN {X 0,Y 256.254,Z 98.952,A -85,B 0,C 180,E1 -18597.642,E2 -18597.642} C_VEL
LIN {X 0,Y 257.767,Z 101.839,A -85,B 0,C 180,E1 -18597.99,E2 -18597.99} C_VEL
LIN {X 0,Y 266.196,Z 117.412,A -85,B 0,C 180,E1 -18599.605,E2 -18599.605} C_VEL
LIN {X 0,Y 272.913,Z 129.611,A -85,B 0,C 180,E1 -18600.796,E2 -18600.796} C_VEL
LIN {X 0,Y 281.844,Z 142.214,A -85,B 0,C 180,E1 -18602.171,E2 -18602.171} C_VEL
LIN {X 0,Y 292.785,Z 154.453,A -85,B 0,C 180,E1 -18603.634,E2 -18603.634} C_VEL
LIN {X 0,Y 304.529,Z 165.897,A -85,B 0,C 180,E1 -18605.074,E2 -18605.074} C_VEL
LIN {X 0,Y 313.787,Z 174.116,A -85,B 0,C 180,E1 -18606.365,E2 -18606.365} C_VEL
LIN {X 0,Y 322.432,Z 181.614,A -85,B 0,C 180,E1 -18607.785,E2 -18607.785} C_VEL
LIN {X 0,Y 331.11,Z 188.727,A -85,B 0,C 180,E1 -18609.427,E2 -18609.427} C_VEL
LIN {X 0,Y 338.95,Z 194.707,A -85,B 0,C 180,E1 -18611.087,E2 -18611.087} C_VEL
LIN {X 0,Y 345.612,Z 199.807,A -85,B 0,C 180,E1 -18612.652,E2 -18612.652} C_VEL
LIN {X 0,Y 351.185,Z 203.799,A -85,B 0,C 180,E1 -18614.103,E2 -18614.103} C_VEL
LIN {X 0,Y 356.383,Z 207.705,A -85,B 0,C 180,E1 -18615.608,E2 -18615.608} C_VEL
LIN {X 0,Y 361.383,Z 210.752,A -85,B 0,C 180,E1 -18617.183,E2 -18617.183} C_VEL
LIN {X 0,Y 364.769,Z 212.87,A -85,B 0,C 180,E1 -18618.404,E2 -18618.404} C_VEL
LIN {X 0,Y 368.888,Z 216.053,A -85,B 0,C 180,E1 -18620.127,E2 -18620.127} C_VEL
LIN {X 0,Y 372.365,Z 218.281,A -85,B 0,C 180,E1 -18621.851,E2 -18621.851} C_VEL
LIN {X 0,Y 375.376,Z 219.894,A -85,B 0,C 180,E1 -18623.707,E2 -18623.707} C_VEL
LIN {X 0,Y 377.795,Z 220.89,A -85,B 0,C 180,E1 -18625.733,E2 -18625.733} C_VEL
LIN {X 0,Y 379.058,Z 221.314,A -85,B 0,C 180,E1 -18627.294,E2 -18627.294} C_VEL
LIN {X 0,Y 379.738,Z 221.784,A -85,B 0,C 180,E1 -18628.94,E2 -18628.94} C_VEL
LIN {X 0,Y 379.893,Z 221.671,A -85,B 0,C 180,E1 -18630,E2 -18630} C_VEL
LIN {X 0,Y 379.625,Z 221.63,A -85,B 0,C 180,E1 -18631.43,E2 -18631.43} C_VEL
LIN {X 0,Y 378.723,Z 221.103,A -85,B 0,C 180,E1 -18633.191,E2 -18633.191} C_VEL
LIN {X 0,Y 376.928,Z 220.57,A -85,B 0,C 180,E1 -18635.077,E2 -18635.077} C_VEL
LIN {X 0,Y 374.242,Z 219.319,A -85,B 0,C 180,E1 -18637.04,E2 -18637.04} C_VEL
LIN {X 0,Y 370.773,Z 217.317,A -85,B 0,C 180,E1 -18638.978,E2 -18638.978} C_VEL
LIN {X 0,Y 366.764,Z 214.51,A -85,B 0,C 180,E1 -18640.79,E2 -18640.79} C_VEL
LIN {X 0,Y 363.238,Z 211.735,A -85,B 0,C 180,E1 -18642.174,E2 -18642.174} C_VEL
LIN {X 0,Y 358.365,Z 208.945,A -85,B 0,C 180,E1 -18643.8,E2 -18643.8} C_VEL
LIN {X 0,Y 352.463,Z 204.842,A -85,B 0,C 180,E1 -18645.538,E2 -18645.538} C_VEL
LIN {X 0,Y 347.439,Z 201.044,A -85,B 0,C 180,E1 -18646.883,E2 -18646.883} C_VEL
LIN {X 0,Y 340.856,Z 196.307,A -85,B 0,C 180,E1 -18648.478,E2 -18648.478} C_VEL
LIN {X 0,Y 334.549,Z 191.341,A -85,B 0,C 180,E1 -18649.868,E2 -18649.868} C_VEL
LIN {X 0,Y 327.42,Z 185.632,A -85,B 0,C 180,E1 -18651.303,E2 -18651.303} C_VEL
LIN {X 0,Y 319.004,Z 178.738,A -85,B 0,C 180,E1 -18652.799,E2 -18652.799} C_VEL
LIN {X 0,Y 311.293,Z 171.971,A -85,B 0,C 180,E1 -18654.001,E2 -18654.001} C_VEL
LIN {X 0,Y 302.062,Z 163.648,A -85,B 0,C 180,E1 -18655.238,E2 -18655.238} C_VEL
LIN {X 0,Y 288.257,Z 149.659,A -85,B 0,C 180,E1 -18656.948,E2 -18656.948} C_VEL
LIN {X 0,Y 279.297,Z 138.876,A -85,B 0,C 180,E1 -18658.203,E2 -18658.203} C_VEL
LIN {X 0,Y 271.488,Z 127.257,A -85,B 0,C 180,E1 -18659.443,E2 -18659.443} C_VEL
LIN {X 0,Y 259.575,Z 105.126,A -85,B 0,C 180,E1 -18661.654,E2 -18661.654} C_VEL
LIN {X 0,Y 256.313,Z 99.12,A -85,B 0,C 180,E1 -18662.334,E2 -18662.334} C_VEL
LIN {X 0,Y 256.097,Z 98.151,A -85,B 0,C 180,E1 -18662.698,E2 -18662.698} C_VEL
LIN {X 0,Y 256.117,Z 98.043,A -85,B 0,C 180,E1 -18665.187,E2 -18665.187} C_VEL
LIN {X 0,Y 256.084,Z 98.067,A -85,B 0,C 180,E1 -18669.14,E2 -18669.14} C_VEL
LIN {X 0,Y 256.046,Z 98.037,A -85,B 0,C 180,E1 -18673.33,E2 -18673.33} C_VEL
LIN {X 0,Y 256.079,Z 98.079,A -85,B 0,C 180,E1 -18677.817,E2 -18677.817} C_VEL
LIN {X 0,Y 256.097,Z 98.076,A -85,B 0,C 180,E1 -18680.864,E2 -18680.864} C_VEL
LIN {X 0,Y 256.119,Z 98.06,A -85,B 0,C 180,E1 -18684.814,E2 -18684.814} C_VEL
LIN {X 0,Y 256.09,Z 98.086,A -85,B 0,C 180,E1 -18688.573,E2 -18688.573} C_VEL
LIN {X 0,Y 256.136,Z 98.05,A -85,B 0,C 180,E1 -18692.197,E2 -18692.197} C_VEL
LIN {X 0,Y 256.166,Z 98.074,A -85,B 0,C 180,E1 -18695.7,E2 -18695.7} C_VEL
LIN {X 0,Y 256.165,Z 98.055,A -85,B 0,C 180,E1 -18699.106,E2 -18699.106} C_VEL
LIN {X 0,Y 256.299,Z 98.053,A -85,B 0,C 180,E1 -18704.086,E2 -18704.086} C_VEL
LIN {X 0,Y 256.31,Z 98.023,A -85,B 0,C 180,E1 -18708.935,E2 -18708.935} C_VEL
LIN {X 0,Y 256.54,Z 98.005,A -85,B 0,C 180,E1 -18712.128,E2 -18712.128} C_VEL
LIN {X 0,Y 256.714,Z 97.974,A -85,B 0,C 180,E1 -18718.432,E2 -18718.432} C_VEL
LIN {X 0,Y 256.714,Z 97.977,A -85,B 0,C 180,E1 -18721.57,E2 -18721.57} C_VEL
LIN {X 0,Y 256.541,Z 98.002,A -85,B 0,C 180,E1 -18727.874,E2 -18727.874} C_VEL
LIN {X 0,Y 256.311,Z 98.023,A -85,B 0,C 180,E1 -18731.067,E2 -18731.067} C_VEL
LIN {X 0,Y 256.301,Z 98.048,A -85,B 0,C 180,E1 -18735.916,E2 -18735.916} C_VEL
LIN {X 0,Y 256.168,Z 98.056,A -85,B 0,C 180,E1 -18740.896,E2 -18740.896} C_VEL
LIN {X 0,Y 256.19,Z 98.055,A -85,B 0,C 180,E1 -18745.139,E2 -18745.139} C_VEL
LIN {X 0,Y 256.105,Z 98.077,A -85,B 0,C 180,E1 -18749.602,E2 -18749.602} C_VEL
LIN {X 0,Y 256.069,Z 98.066,A -85,B 0,C 180,E1 -18753.293,E2 -18753.293} C_VEL
LIN {X 0,Y 256.117,Z 98.083,A -85,B 0,C 180,E1 -18757.272,E2 -18757.272} C_VEL
LIN {X 0,Y 256.056,Z 98.077,A -85,B 0,C 180,E1 -18761.204,E2 -18761.204} C_VEL
LIN {X 0,Y 256.043,Z 98.082,A -85,B 0,C 180,E1 -18765.535,E2 -18765.535} C_VEL
LIN {X 0,Y 256.043,Z 98.087,A -85,B 0,C 180,E1 -18766.196,E2 -18766.196} C_VEL
LIN {X 0,Y 255.346,Z 98.192,A -85,B 0,C 180,E1 -18767.088,E2 -18767.088} C_VEL
LIN {X 0,Y 252.407,Z 98.517,A -85,B 0,C 180,E1 -18768.489,E2 -18768.489} C_VEL
LIN {X 0,Y 249.673,Z 98.967,A -85,B 0,C 180,E1 -18769.89,E2 -18769.89} C_VEL
LIN {X 0,Y 249.223,Z 99.738,A -85,B 0,C 180,E1 -18770.614,E2 -18770.614} C_VEL
LIN {X 0,Y 249.261,Z 99.968,A -85,B 0,C 180,E1 -18770.755,E2 -18770.755} C_VEL
LIN {X 0,Y 250.61,Z 105.701,A -85,B 0,C 180,E1 -18773.92,E2 -18773.92} C_VEL
LIN {X 0,Y 251.81,Z 111.656,A -85,B 0,C 180,E1 -18776.982,E2 -18776.982} C_VEL
LIN {X 0,Y 253.258,Z 115.242,A -85,B 0,C 180,E1 -18777.41,E2 -18777.41} C_VEL
LIN {X 0,Y 260.484,Z 131.638,A -85,B 0,C 180,E1 -18778.931,E2 -18778.931} C_VEL
LIN {X 0,Y 263.149,Z 143.621,A -85,B 0,C 180,E1 -18779.648,E2 -18779.648} C_VEL
LIN {X 0,Y 266.541,Z 163.261,A -85,B 0,C 180,E1 -18780.666,E2 -18780.666} C_VEL
LIN {X 0,Y 264.853,Z 217.518,A -85,B 0,C 180,E1 -18782.149,E2 -18782.149} C_VEL
LIN {X 0,Y 264.108,Z 227.668,A -85,B 0,C 180,E1 -18782.585,E2 -18782.585} C_VEL
LIN {X 0,Y 263.129,Z 236.495,A -85,B 0,C 180,E1 -18783.103,E2 -18783.103} C_VEL
LIN {X 0,Y 261.906,Z 245.848,A -85,B 0,C 180,E1 -18783.827,E2 -18783.827} C_VEL
LIN {X 0,Y 260.305,Z 255.985,A -85,B 0,C 180,E1 -18784.835,E2 -18784.835} C_VEL
LIN {X 0,Y 258.625,Z 264.977,A -85,B 0,C 180,E1 -18785.945,E2 -18785.945} C_VEL
LIN {X 0,Y 256.874,Z 273.702,A -85,B 0,C 180,E1 -18787.266,E2 -18787.266} C_VEL
LIN {X 0,Y 255.276,Z 281.094,A -85,B 0,C 180,E1 -18788.606,E2 -18788.606} C_VEL
LIN {X 0,Y 253.629,Z 288.311,A -85,B 0,C 180,E1 -18790.157,E2 -18790.157} C_VEL
LIN {X 0,Y 252.449,Z 294.107,A -85,B 0,C 180,E1 -18791.623,E2 -18791.623} C_VEL
LIN {X 0,Y 250.767,Z 301.052,A -85,B 0,C 180,E1 -18793.724,E2 -18793.724} C_VEL
LIN {X 0,Y 249.7,Z 305.553,A -85,B 0,C 180,E1 -18795.326,E2 -18795.326} C_VEL
LIN {X 0,Y 248.418,Z 311.044,A -85,B 0,C 180,E1 -18797.75,E2 -18797.75} C_VEL
LIN {X 0,Y 247.614,Z 315.373,A -85,B 0,C 180,E1 -18800.195,E2 -18800.195} C_VEL
LIN {X 0,Y 247.262,Z 317.743,A -85,B 0,C 180,E1 -18801.83,E2 -18801.83} C_VEL
LIN {X 0,Y 247.011,Z 319.544,A -85,B 0,C 180,E1 -18803.465,E2 -18803.465} C_VEL
LIN {X 0,Y 246.855,Z 321.996,A -85,B 0,C 180,E1 -18806.736,E2 -18806.736} C_VEL
LIN {X 0,Y 246.904,Z 322.589,A -85,B 0,C 180,E1 -18808.369,E2 -18808.369} C_VEL
LIN {X 0,Y 246.983,Z 322.746,A -85,B 0,C 180,E1 -18810,E2 -18810} C_VEL
LIN {X 0,Y 246.904,Z 322.589,A -85,B 0,C 180,E1 -18811.631,E2 -18811.631} C_VEL
LIN {X 0,Y 246.855,Z 321.996,A -85,B 0,C 180,E1 -18813.264,E2 -18813.264} C_VEL
LIN {X 0,Y 247.011,Z 319.544,A -85,B 0,C 180,E1 -18816.535,E2 -18816.535} C_VEL
LIN {X 0,Y 247.411,Z 316.591,A -85,B 0,C 180,E1 -18818.988,E2 -18818.988} C_VEL
LIN {X 0,Y 248.116,Z 312.6,A -85,B 0,C 180,E1 -18821.436,E2 -18821.436} C_VEL
LIN {X 0,Y 249.192,Z 307.468,A -85,B 0,C 180,E1 -18823.87,E2 -18823.87} C_VEL
LIN {X 0,Y 250.506,Z 302.208,A -85,B 0,C 180,E1 -18825.875,E2 -18825.875} C_VEL
LIN {X 0,Y 252.007,Z 295.892,A -85,B 0,C 180,E1 -18827.865,E2 -18827.865} C_VEL
LIN {X 0,Y 253.709,Z 288.314,A -85,B 0,C 180,E1 -18829.836,E2 -18829.836} C_VEL
LIN {X 0,Y 255.708,Z 279.175,A -85,B 0,C 180,E1 -18831.78,E2 -18831.78} C_VEL
LIN {X 0,Y 258.12,Z 267.679,A -85,B 0,C 180,E1 -18833.679,E2 -18833.679} C_VEL
LIN {X 0,Y 260.026,Z 257.616,A -85,B 0,C 180,E1 -18834.981,E2 -18834.981} C_VEL
LIN {X 0,Y 261.577,Z 247.86,A -85,B 0,C 180,E1 -18835.994,E2 -18835.994} C_VEL
LIN {X 0,Y 262.799,Z 239.069,A -85,B 0,C 180,E1 -18836.719,E2 -18836.719} C_VEL
LIN {X 0,Y 263.968,Z 228.522,A -85,B 0,C 180,E1 -18837.378,E2 -18837.378} C_VEL
LIN {X 0,Y 264.732,Z 218.77,A -85,B 0,C 180,E1 -18837.811,E2 -18837.811} C_VEL
LIN {X 0,Y 265.813,Z 189.042,A -85,B 0,C 180,E1 -18838.642,E2 -18838.642} C_VEL
LIN {X 0,Y 266.542,Z 163.25,A -85,B 0,C 180,E1 -18839.334,E2 -18839.334} C_VEL
LIN {X 0,Y 262.742,Z 141.781,A -85,B 0,C 180,E1 -18840.46,E2 -18840.46} C_VEL
LIN {X 0,Y 260.498,Z 131.702,A -85,B 0,C 180,E1 -18841.065,E2 -18841.065} C_VEL
LIN {X 0,Y 253.278,Z 115.225,A -85,B 0,C 180,E1 -18842.587,E2 -18842.587} C_VEL
LIN {X 0,Y 251.852,Z 111.848,A -85,B 0,C 180,E1 -18842.968,E2 -18842.968} C_VEL
LIN {X 0,Y 250.603,Z 105.701,A -85,B 0,C 180,E1 -18846.081,E2 -18846.081} C_VEL
LIN {X 0,Y 249.099,Z 99.23,A -85,B 0,C 180,E1 -18849.668,E2 -18849.668} C_VEL
LIN {X 0,Y 249.028,Z 98.93,A -85,B 0,C 180,E1 -18850.474,E2 -18850.474} C_VEL
LIN {X 0,Y 248.988,Z 98.959,A -85,B 0,C 180,E1 -18854.882,E2 -18854.882} C_VEL
LIN {X 0,Y 249.012,Z 98.971,A -85,B 0,C 180,E1 -18857.361,E2 -18857.361} C_VEL
LIN {X 0,Y 249.028,Z 98.96,A -85,B 0,C 180,E1 -18861.619,E2 -18861.619} C_VEL
LIN {X 0,Y 249.045,Z 98.936,A -85,B 0,C 180,E1 -18865.639,E2 -18865.639} C_VEL
LIN {X 0,Y 249.049,Z 98.962,A -85,B 0,C 180,E1 -18869.472,E2 -18869.472} C_VEL
LIN {X 0,Y 249.073,Z 98.926,A -85,B 0,C 180,E1 -18873.161,E2 -18873.161} C_VEL
LIN {X 0,Y 249.081,Z 98.958,A -85,B 0,C 180,E1 -18876.732,E2 -18876.732} C_VEL
LIN {X 0,Y 249.111,Z 98.917,A -85,B 0,C 180,E1 -18880.211,E2 -18880.211} C_VEL
LIN {X 0,Y 249.243,Z 98.921,A -85,B 0,C 180,E1 -18883.621,E2 -18883.621} C_VEL
LIN {X 0,Y 249.254,Z 98.905,A -85,B 0,C 180,E1 -18888.616,E2 -18888.616} C_VEL
LIN {X 0,Y 249.483,Z 98.876,A -85,B 0,C 180,E1 -18891.902,E2 -18891.902} C_VEL
LIN {X 0,Y 249.436,Z 98.907,A -85,B 0,C 180,E1 -18896.769,E2 -18896.769} C_VEL
LIN {X 0,Y 249.721,Z 98.833,A -85,B 0,C 180,E1 -18899.999,E2 -18899.999} C_VEL
LIN {X 0,Y 249.436,Z 98.905,A -85,B 0,C 180,E1 -18903.23,E2 -18903.23} C_VEL
LIN {X 0,Y 249.481,Z 98.879,A -85,B 0,C 180,E1 -18908.096,E2 -18908.096} C_VEL
LIN {X 0,Y 249.253,Z 98.905,A -85,B 0,C 180,E1 -18911.383,E2 -18911.383} C_VEL
LIN {X 0,Y 249.241,Z 98.927,A -85,B 0,C 180,E1 -18916.377,E2 -18916.377} C_VEL
LIN {X 0,Y 249.086,Z 98.945,A -85,B 0,C 180,E1 -18921.517,E2 -18921.517} C_VEL
LIN {X 0,Y 249.129,Z 98.935,A -85,B 0,C 180,E1 -18925.481,E2 -18925.481} C_VEL
LIN {X 0,Y 249.071,Z 98.942,A -85,B 0,C 180,E1 -18928.988,E2 -18928.988} C_VEL
LIN {X 0,Y 249.034,Z 98.956,A -85,B 0,C 180,E1 -18932.424,E2 -18932.424} C_VEL
LIN {X 0,Y 249.072,Z 98.951,A -85,B 0,C 180,E1 -18936.337,E2 -18936.337} C_VEL
LIN {X 0,Y 249.031,Z 98.945,A -85,B 0,C 180,E1 -18940.472,E2 -18940.472} C_VEL
LIN {X 0,Y 248.994,Z 98.949,A -85,B 0,C 180,E1 -18944.88,E2 -18944.88} C_VEL
LIN {X 0,Y 249.006,Z 98.907,A -85,B 0,C 180,E1 -18947.361,E2 -18947.361} C_VEL
LIN {X 0,Y 249.035,Z 98.963,A -85,B 0,C 180,E1 -18951.621,E2 -18951.621} C_VEL
LIN {X 0,Y 249.058,Z 98.921,A -85,B 0,C 180,E1 -18955.642,E2 -18955.642} C_VEL
LIN {X 0,Y 249.07,Z 99.185,A -85,B 0,C 180,E1 -18956.444,E2 -18956.444} C_VEL
LIN {X 0,Y 249.428,Z 100.508,A -85,B 0,C 180,E1 -18956.719,E2 -18956.719} C_VEL
LIN {X 0,Y 258.476,Z 116.687,A -85,B 0,C 180,E1 -18958.565,E2 -18958.565} C_VEL
LIN {X 0,Y 267.406,Z 133.35,A -85,B 0,C 180,E1 -18960.243,E2 -18960.243} C_VEL
LIN {X 0,Y 276.27,Z 146.094,A -85,B 0,C 180,E1 -18961.667,E2 -18961.667} C_VEL
LIN {X 0,Y 286.44,Z 157.731,A -85,B 0,C 180,E1 -18963.088,E2 -18963.088} C_VEL
LIN {X 0,Y 299.644,Z 170.838,A -85,B 0,C 180,E1 -18964.719,E2 -18964.719} C_VEL
LIN {X 0,Y 308.969,Z 179.069,A -85,B 0,C 180,E1 -18965.923,E2 -18965.923} C_VEL
LIN {X 0,Y 316.903,Z 185.851,A -85,B 0,C 180,E1 -18967.117,E2 -18967.117} C_VEL
LIN {X 0,Y 323.841,Z 191.356,A -85,B 0,C 180,E1 -18968.297,E2 -18968.297} C_VEL
LIN {X 0,Y 330.666,Z 196.835,A -85,B 0,C 180,E1 -18969.595,E2 -18969.595} C_VEL
LIN {X 0,Y 337.791,Z 202.22,A -85,B 0,C 180,E1 -18971.097,E2 -18971.097} C_VEL
LIN {X 0,Y 344.657,Z 207.219,A -85,B 0,C 180,E1 -18972.691,E2 -18972.691} C_VEL
LIN {X 0,Y 351.097,Z 211.927,A -85,B 0,C 180,E1 -18974.381,E2 -18974.381} C_VEL
LIN {X 0,Y 356.33,Z 215.555,A -85,B 0,C 180,E1 -18975.904,E2 -18975.904} C_VEL
LIN {X 0,Y 361.308,Z 218.368,A -85,B 0,C 180,E1 -18977.496,E2 -18977.496} C_VEL
LIN {X 0,Y 366.147,Z 221.933,A -85,B 0,C 180,E1 -18979.35,E2 -18979.35} C_VEL
LIN {X 0,Y 370.063,Z 224.603,A -85,B 0,C 180,E1 -18981.161,E2 -18981.161} C_VEL
LIN {X 0,Y 373.324,Z 226.403,A -85,B 0,C 180,E1 -18982.996,E2 -18982.996} C_VEL
LIN {X 0,Y 375.946,Z 227.609,A -85,B 0,C 180,E1 -18984.91,E2 -18984.91} C_VEL
LIN {X 0,Y 377.765,Z 228.134,A -85,B 0,C 180,E1 -18986.801,E2 -18986.801} C_VEL
LIN {X 0,Y 378.667,Z 228.708,A -85,B 0,C 180,E1 -18988.581,E2 -18988.581} C_VEL
LIN {X 0,Y 378.931,Z 228.683,A -85,B 0,C 180,E1 -18990,E2 -18990} C_VEL
LIN {X 0,Y 378.671,Z 228.665,A -85,B 0,C 180,E1 -18991.434,E2 -18991.434} C_VEL
LIN {X 0,Y 377.771,Z 228.117,A -85,B 0,C 180,E1 -18993.199,E2 -18993.199} C_VEL
LIN {X 0,Y 375.952,Z 227.604,A -85,B 0,C 180,E1 -18995.091,E2 -18995.091} C_VEL
LIN {X 0,Y 373.246,Z 226.355,A -85,B 0,C 180,E1 -18997.059,E2 -18997.059} C_VEL
LIN {X 0,Y 369.756,Z 224.393,A -85,B 0,C 180,E1 -18999,E2 -18999} C_VEL
LIN {X 0,Y 365.721,Z 221.637,A -85,B 0,C 180,E1 -19000.821,E2 -19000.821} C_VEL
LIN {X 0,Y 361.434,Z 218.445,A -85,B 0,C 180,E1 -19002.46,E2 -19002.46} C_VEL
LIN {X 0,Y 356.574,Z 215.656,A -85,B 0,C 180,E1 -19004.026,E2 -19004.026} C_VEL
LIN {X 0,Y 351.283,Z 212.07,A -85,B 0,C 180,E1 -19005.567,E2 -19005.567} C_VEL
LIN {X 0,Y 345.254,Z 207.593,A -85,B 0,C 180,E1 -19007.157,E2 -19007.157} C_VEL
LIN {X 0,Y 337.822,Z 202.302,A -85,B 0,C 180,E1 -19008.895,E2 -19008.895} C_VEL
LIN {X 0,Y 331.928,Z 197.735,A -85,B 0,C 180,E1 -19010.15,E2 -19010.15} C_VEL
LIN {X 0,Y 325.338,Z 192.633,A -85,B 0,C 180,E1 -19011.424,E2 -19011.424} C_VEL
LIN {X 0,Y 317.858,Z 186.627,A -85,B 0,C 180,E1 -19012.731,E2 -19012.731} C_VEL
LIN {X 0,Y 309.933,Z 179.873,A -85,B 0,C 180,E1 -19013.942,E2 -19013.942} C_VEL
LIN {X 0,Y 302.076,Z 172.929,A -85,B 0,C 180,E1 -19014.988,E2 -19014.988} C_VEL
LIN {X 0,Y 293.956,Z 165.319,A -85,B 0,C 180,E1 -19015.962,E2 -19015.962} C_VEL
LIN {X 0,Y 283.333,Z 154.443,A -85,B 0,C 180,E1 -19017.326,E2 -19017.326} C_VEL
LIN {X 0,Y 274.531,Z 143.799,A -85,B 0,C 180,E1 -19018.598,E2 -19018.598} C_VEL
LIN {X 0,Y 266.339,Z 131.557,A -85,B 0,C 180,E1 -19019.944,E2 -19019.944} C_VEL
LIN {X 0,Y 254.283,Z 109.024,A -85,B 0,C 180,E1 -19022.269,E2 -19022.269} C_VEL
LIN {X 0,Y 250.277,Z 102.168,A -85,B 0,C 180,E1 -19023.085,E2 -19023.085} C_VEL
LIN {X 0,Y 249.139,Z 99.551,A -85,B 0,C 180,E1 -19023.441,E2 -19023.441} C_VEL
LIN {X 0,Y 249.044,Z 98.988,A -85,B 0,C 180,E1 -19023.777,E2 -19023.777} C_VEL
LIN {X 0,Y 249.052,Z 98.964,A -85,B 0,C 180,E1 -19027.804,E2 -19027.804} C_VEL
LIN {X 0,Y 249.022,Z 98.915,A -85,B 0,C 180,E1 -19030.475,E2 -19030.475} C_VEL
LIN {X 0,Y 248.992,Z 98.944,A -85,B 0,C 180,E1 -19034.882,E2 -19034.882} C_VEL
LIN {X 0,Y 249.021,Z 98.963,A -85,B 0,C 180,E1 -19037.365,E2 -19037.365} C_VEL
LIN {X 0,Y 249.045,Z 98.962,A -85,B 0,C 180,E1 -19041.624,E2 -19041.624} C_VEL
LIN {X 0,Y 249.059,Z 98.936,A -85,B 0,C 180,E1 -19045.643,E2 -19045.643} C_VEL
LIN {X 0,Y 249.045,Z 98.962,A -85,B 0,C 180,E1 -19049.473,E2 -19049.473} C_VEL
LIN {X 0,Y 249.07,Z 98.929,A -85,B 0,C 180,E1 -19053.163,E2 -19053.163} C_VEL
LIN {X 0,Y 249.078,Z 98.961,A -85,B 0,C 180,E1 -19056.734,E2 -19056.734} C_VEL
LIN {X 0,Y 249.108,Z 98.919,A -85,B 0,C 180,E1 -19060.212,E2 -19060.212} C_VEL
LIN {X 0,Y 249.241,Z 98.927,A -85,B 0,C 180,E1 -19063.623,E2 -19063.623} C_VEL
LIN {X 0,Y 249.253,Z 98.905,A -85,B 0,C 180,E1 -19068.617,E2 -19068.617} C_VEL
LIN {X 0,Y 249.481,Z 98.879,A -85,B 0,C 180,E1 -19071.904,E2 -19071.904} C_VEL
LIN {X 0,Y 249.436,Z 98.905,A -85,B 0,C 180,E1 -19076.77,E2 -19076.77} C_VEL
LIN {X 0,Y 249.721,Z 98.833,A -85,B 0,C 180,E1 -19080.001,E2 -19080.001} C_VEL
LIN {X 0,Y 249.436,Z 98.907,A -85,B 0,C 180,E1 -19083.231,E2 -19083.231} C_VEL
LIN {X 0,Y 249.483,Z 98.876,A -85,B 0,C 180,E1 -19088.098,E2 -19088.098} C_VEL
LIN {X 0,Y 249.254,Z 98.905,A -85,B 0,C 180,E1 -19091.384,E2 -19091.384} C_VEL
LIN {X 0,Y 249.243,Z 98.921,A -85,B 0,C 180,E1 -19096.379,E2 -19096.379} C_VEL
LIN {X 0,Y 249.089,Z 98.945,A -85,B 0,C 180,E1 -19101.519,E2 -19101.519} C_VEL
LIN {X 0,Y 249.132,Z 98.93,A -85,B 0,C 180,E1 -19105.483,E2 -19105.483} C_VEL
LIN {X 0,Y 249.075,Z 98.945,A -85,B 0,C 180,E1 -19108.99,E2 -19108.99} C_VEL
LIN {X 0,Y 249.032,Z 98.952,A -85,B 0,C 180,E1 -19112.427,E2 -19112.427} C_VEL
LIN {X 0,Y 249.05,Z 98.957,A -85,B 0,C 180,E1 -19116.343,E2 -19116.343} C_VEL
LIN {X 0,Y 249.008,Z 98.95,A -85,B 0,C 180,E1 -19120.479,E2 -19120.479} C_VEL
LIN {X 0,Y 248.988,Z 98.958,A -85,B 0,C 180,E1 -19124.884,E2 -19124.884} C_VEL
LIN {X 0,Y 249.018,Z 98.959,A -85,B 0,C 180,E1 -19127.363,E2 -19127.363} C_VEL
LIN {X 0,Y 249.051,Z 99.047,A -85,B 0,C 180,E1 -19130.192,E2 -19130.192} C_VEL
LIN {X 0,Y 249.261,Z 99.968,A -85,B 0,C 180,E1 -19130.755,E2 -19130.755} C_VEL
LIN {X 0,Y 248.99,Z 101.639,A -85,B 0,C 180,E1 -19131.579,E2 -19131.579} C_VEL
LIN {X 0,Y 246.798,Z 104.784,A -85,B 0,C 180,E1 -19132.855,E2 -19132.855} C_VEL
LIN {X 0,Y 244.524,Z 107.942,A -85,B 0,C 180,E1 -19134.153,E2 -19134.153} C_VEL
LIN {X 0,Y 244.161,Z 109.654,A -85,B 0,C 180,E1 -19134.999,E2 -19134.999} C_VEL
LIN {X 0,Y 244.572,Z 111.681,A -85,B 0,C 180,E1 -19135.928,E2 -19135.928} C_VEL
LIN {X 0,Y 250.497,Z 124.588,A -85,B 0,C 180,E1 -19137.32,E2 -19137.32} C_VEL
LIN {X 0,Y 255.102,Z 135.444,A -85,B 0,C 180,E1 -19138.328,E2 -19138.328} C_VEL
LIN {X 0,Y 259.195,Z 157.093,A -85,B 0,C 180,E1 -19139.563,E2 -19139.563} C_VEL
LIN {X 0,Y 260.396,Z 165.747,A -85,B 0,C 180,E1 -19139.987,E2 -19139.987} C_VEL
LIN {X 0,Y 258.576,Z 217.97,A -85,B 0,C 180,E1 -19141.44,E2 -19141.44} C_VEL
LIN {X 0,Y 257.735,Z 228.524,A -85,B 0,C 180,E1 -19141.914,E2 -19141.914} C_VEL
LIN {X 0,Y 256.473,Z 238.878,A -85,B 0,C 180,E1 -19142.568,E2 -19142.568} C_VEL
LIN {X 0,Y 254.793,Z 250.691,A -85,B 0,C 180,E1 -19143.591,E2 -19143.591} C_VEL
LIN {X 0,Y 252.715,Z 262.084,A -85,B 0,C 180,E1 -19144.906,E2 -19144.906} C_VEL
LIN {X 0,Y 250.585,Z 272.377,A -85,B 0,C 180,E1 -19146.443,E2 -19146.443} C_VEL
LIN {X 0,Y 248.642,Z 280.903,A -85,B 0,C 180,E1 -19148.006,E2 -19148.006} C_VEL
LIN {X 0,Y 246.932,Z 288.12,A -85,B 0,C 180,E1 -19149.595,E2 -19149.595} C_VEL
LIN {X 0,Y 245.615,Z 294.217,A -85,B 0,C 180,E1 -19151.188,E2 -19151.188} C_VEL
LIN {X 0,Y 243.916,Z 300.86,A -85,B 0,C 180,E1 -19153.254,E2 -19153.254} C_VEL
LIN {X 0,Y 242.806,Z 305.362,A -85,B 0,C 180,E1 -19154.9,E2 -19154.9} C_VEL
LIN {X 0,Y 241.446,Z 310.853,A -85,B 0,C 180,E1 -19157.39,E2 -19157.39} C_VEL
LIN {X 0,Y 240.601,Z 315.182,A -85,B 0,C 180,E1 -19159.906,E2 -19159.906} C_VEL
LIN {X 0,Y 240.209,Z 317.552,A -85,B 0,C 180,E1 -19161.588,E2 -19161.588} C_VEL
LIN {X 0,Y 239.928,Z 319.353,A -85,B 0,C 180,E1 -19163.271,E2 -19163.271} C_VEL
LIN {X 0,Y 239.762,Z 321.806,A -85,B 0,C 180,E1 -19166.639,E2 -19166.639} C_VEL
LIN {X 0,Y 239.816,Z 322.399,A -85,B 0,C 180,E1 -19168.321,E2 -19168.321} C_VEL
LIN {X 0,Y 239.891,Z 322.556,A -85,B 0,C 180,E1 -19170,E2 -19170} C_VEL
LIN {X 0,Y 239.816,Z 322.399,A -85,B 0,C 180,E1 -19171.679,E2 -19171.679} C_VEL
LIN {X 0,Y 239.761,Z 321.806,A -85,B 0,C 180,E1 -19173.361,E2 -19173.361} C_VEL
LIN {X 0,Y 239.928,Z 319.353,A -85,B 0,C 180,E1 -19176.729,E2 -19176.729} C_VEL
LIN {X 0,Y 240.377,Z 316.4,A -85,B 0,C 180,E1 -19179.254,E2 -19179.254} C_VEL
LIN {X 0,Y 241.138,Z 312.408,A -85,B 0,C 180,E1 -19181.772,E2 -19181.772} C_VEL
LIN {X 0,Y 242.28,Z 307.277,A -85,B 0,C 180,E1 -19184.274,E2 -19184.274} C_VEL
LIN {X 0,Y 243.657,Z 302.017,A -85,B 0,C 180,E1 -19186.333,E2 -19186.333} C_VEL
LIN {X 0,Y 245.235,Z 295.701,A -85,B 0,C 180,E1 -19188.375,E2 -19188.375} C_VEL
LIN {X 0,Y 246.638,Z 289.749,A -85,B 0,C 180,E1 -19189.995,E2 -19189.995} C_VEL
LIN {X 0,Y 248.202,Z 282.821,A -85,B 0,C 180,E1 -19191.599,E2 -19191.599} C_VEL
LIN {X 0,Y 250.119,Z 274.647,A -85,B 0,C 180,E1 -19193.165,E2 -19193.165} C_VEL
LIN {X 0,Y 251.917,Z 266.138,A -85,B 0,C 180,E1 -19194.518,E2 -19194.518} C_VEL
LIN {X 0,Y 253.594,Z 257.426,A -85,B 0,C 180,E1 -19195.66,E2 -19195.66} C_VEL
LIN {X 0,Y 255.222,Z 247.67,A -85,B 0,C 180,E1 -19196.692,E2 -19196.692} C_VEL
LIN {X 0,Y 256.494,Z 238.879,A -85,B 0,C 180,E1 -19197.43,E2 -19197.43} C_VEL
LIN {X 0,Y 257.663,Z 228.533,A -85,B 0,C 180,E1 -19198.094,E2 -19198.094} C_VEL
LIN {X 0,Y 258.517,Z 217.974,A -85,B 0,C 180,E1 -19198.566,E2 -19198.566} C_VEL
LIN {X 0,Y 260.361,Z 164.299,A -85,B 0,C 180,E1 -19200.062,E2 -19200.062} C_VEL
LIN {X 0,Y 256.747,Z 143.662,A -85,B 0,C 180,E1 -19201.184,E2 -19201.184} C_VEL
LIN {X 0,Y 254.684,Z 134.403,A -85,B 0,C 180,E1 -19201.763,E2 -19201.763} C_VEL
LIN {X 0,Y 247.868,Z 118.845,A -85,B 0,C 180,E1 -19203.262,E2 -19203.262} C_VEL
LIN {X 0,Y 244.646,Z 111.857,A -85,B 0,C 180,E1 -19204.035,E2 -19204.035} C_VEL
LIN {X 0,Y 244.338,Z 110.569,A -85,B 0,C 180,E1 -19204.507,E2 -19204.507} C_VEL
LIN {X 0,Y 243.082,Z 104.372,A -85,B 0,C 180,E1 -19207.969,E2 -19207.969} C_VEL
LIN {X 0,Y 241.995,Z 99.882,A -85,B 0,C 180,E1 -19210.669,E2 -19210.669} C_VEL
LIN {X 0,Y 241.923,Z 99.843,A -85,B 0,C 180,E1 -19214.204,E2 -19214.204} C_VEL
LIN {X 0,Y 241.936,Z 99.845,A -85,B 0,C 180,E1 -19218.076,E2 -19218.076} C_VEL
LIN {X 0,Y 241.992,Z 99.842,A -85,B 0,C 180,E1 -19222.418,E2 -19222.418} C_VEL
LIN {X 0,Y 241.982,Z 99.818,A -85,B 0,C 180,E1 -19226.507,E2 -19226.507} C_VEL
LIN {X 0,Y 242.015,Z 99.828,A -85,B 0,C 180,E1 -19230.596,E2 -19230.596} C_VEL
LIN {X 0,Y 242.069,Z 99.804,A -85,B 0,C 180,E1 -19234.182,E2 -19234.182} C_VEL
LIN {X 0,Y 242.055,Z 99.823,A -85,B 0,C 180,E1 -19238.296,E2 -19238.296} C_VEL
LIN {X 0,Y 242.165,Z 99.795,A -85,B 0,C 180,E1 -19243.277,E2 -19243.277} C_VEL
LIN {X 0,Y 242.188,Z 99.79,A -85,B 0,C 180,E1 -19248.279,E2 -19248.279} C_VEL
LIN {X 0,Y 242.429,Z 99.75,A -85,B 0,C 180,E1 -19251.665,E2 -19251.665} C_VEL
LIN {X 0,Y 242.262,Z 99.807,A -85,B 0,C 180,E1 -19255.006,E2 -19255.006} C_VEL
LIN {X 0,Y 242.636,Z 99.729,A -85,B 0,C 180,E1 -19258.339,E2 -19258.339} C_VEL
LIN {X 0,Y 242.636,Z 99.726,A -85,B 0,C 180,E1 -19261.659,E2 -19261.659} C_VEL
LIN {X 0,Y 242.43,Z 99.777,A -85,B 0,C 180,E1 -19266.716,E2 -19266.716} C_VEL
LIN {X 0,Y 242.314,Z 99.757,A -85,B 0,C 180,E1 -19270.021,E2 -19270.021} C_VEL
LIN {X 0,Y 242.167,Z 99.82,A -85,B 0,C 180,E1 -19275.14,E2 -19275.14} C_VEL
LIN {X 0,Y 242.072,Z 99.793,A -85,B 0,C 180,E1 -19278.623,E2 -19278.623} C_VEL
LIN {X 0,Y 242.012,Z 99.835,A -85,B 0,C 180,E1 -19282.179,E2 -19282.179} C_VEL
LIN {X 0,Y 242.065,Z 99.809,A -85,B 0,C 180,E1 -19285.837,E2 -19285.837} C_VEL
LIN {X 0,Y 242.005,Z 99.83,A -85,B 0,C 180,E1 -19289.582,E2 -19289.582} C_VEL
LIN {X 0,Y 241.989,Z 99.821,A -85,B 0,C 180,E1 -19293.49,E2 -19293.49} C_VEL
LIN {X 0,Y 242.009,Z 99.841,A -85,B 0,C 180,E1 -19297.577,E2 -19297.577} C_VEL
LIN {X 0,Y 241.947,Z 99.834,A -85,B 0,C 180,E1 -19301.919,E2 -19301.919} C_VEL
LIN {X 0,Y 241.924,Z 99.794,A -85,B 0,C 180,E1 -19306.572,E2 -19306.572} C_VEL
LIN {X 0,Y 241.969,Z 99.806,A -85,B 0,C 180,E1 -19310.284,E2 -19310.284} C_VEL
LIN {X 0,Y 242.034,Z 99.798,A -85,B 0,C 180,E1 -19314.497,E2 -19314.497} C_VEL
LIN {X 0,Y 242.062,Z 100.089,A -85,B 0,C 180,E1 -19315.369,E2 -19315.369} C_VEL
LIN {X 0,Y 242.424,Z 101.435,A -85,B 0,C 180,E1 -19315.652,E2 -19315.652} C_VEL
LIN {X 0,Y 248.869,Z 112.659,A -85,B 0,C 180,E1 -19317.057,E2 -19317.057} C_VEL
LIN {X 0,Y 256.446,Z 126.945,A -85,B 0,C 180,E1 -19318.616,E2 -19318.616} C_VEL
LIN {X 0,Y 263.309,Z 139.247,A -85,B 0,C 180,E1 -19319.911,E2 -19319.911} C_VEL
LIN {X 0,Y 272.221,Z 151.917,A -85,B 0,C 180,E1 -19321.374,E2 -19321.374} C_VEL
LIN {X 0,Y 282.087,Z 163.106,A -85,B 0,C 180,E1 -19322.786,E2 -19322.786} C_VEL
LIN {X 0,Y 294.898,Z 175.943,A -85,B 0,C 180,E1 -19324.409,E2 -19324.409} C_VEL
LIN {X 0,Y 306.269,Z 185.756,A -85,B 0,C 180,E1 -19325.791,E2 -19325.791} C_VEL
LIN {X 0,Y 315.071,Z 193.147,A -85,B 0,C 180,E1 -19327.073,E2 -19327.073} C_VEL
LIN {X 0,Y 322.412,Z 198.877,A -85,B 0,C 180,E1 -19328.287,E2 -19328.287} C_VEL
LIN {X 0,Y 329.315,Z 204.113,A -85,B 0,C 180,E1 -19329.579,E2 -19329.579} C_VEL
LIN {X 0,Y 337.88,Z 210.642,A -85,B 0,C 180,E1 -19331.388,E2 -19331.388} C_VEL
LIN {X 0,Y 345.549,Z 215.854,A -85,B 0,C 180,E1 -19333.202,E2 -19333.202} C_VEL
LIN {X 0,Y 351.719,Z 220.408,A -85,B 0,C 180,E1 -19334.864,E2 -19334.864} C_VEL
LIN {X 0,Y 357.332,Z 223.941,A -85,B 0,C 180,E1 -19336.571,E2 -19336.571} C_VEL
LIN {X 0,Y 361.256,Z 226.268,A -85,B 0,C 180,E1 -19337.912,E2 -19337.912} C_VEL
LIN {X 0,Y 365.8,Z 229.713,A -85,B 0,C 180,E1 -19339.774,E2 -19339.774} C_VEL
LIN {X 0,Y 369.468,Z 232.044,A -85,B 0,C 180,E1 -19341.544,E2 -19341.544} C_VEL
LIN {X 0,Y 372.781,Z 233.775,A -85,B 0,C 180,E1 -19343.505,E2 -19343.505} C_VEL
LIN {X 0,Y 374.916,Z 234.691,A -85,B 0,C 180,E1 -19345.169,E2 -19345.169} C_VEL
LIN {X 0,Y 376.625,Z 235.242,A -85,B 0,C 180,E1 -19347.059,E2 -19347.059} C_VEL
LIN {X 0,Y 377.427,Z 235.787,A -85,B 0,C 180,E1 -19348.933,E2 -19348.933} C_VEL
LIN {X 0,Y 377.605,Z 235.659,A -85,B 0,C 180,E1 -19350,E2 -19350} C_VEL
LIN {X 0,Y 377.308,Z 235.603,A -85,B 0,C 180,E1 -19351.601,E2 -19351.601} C_VEL
LIN {X 0,Y 376.471,Z 235.083,A -85,B 0,C 180,E1 -19353.21,E2 -19353.21} C_VEL
LIN {X 0,Y 374.597,Z 234.572,A -85,B 0,C 180,E1 -19355.109,E2 -19355.109} C_VEL
LIN {X 0,Y 371.865,Z 233.327,A -85,B 0,C 180,E1 -19357.086,E2 -19357.086} C_VEL
LIN {X 0,Y 368.319,Z 231.356,A -85,B 0,C 180,E1 -19359.035,E2 -19359.035} C_VEL
LIN {X 0,Y 364.355,Z 228.688,A -85,B 0,C 180,E1 -19360.841,E2 -19360.841} C_VEL
LIN {X 0,Y 359.989,Z 225.37,A -85,B 0,C 180,E1 -19362.545,E2 -19362.545} C_VEL
LIN {X 0,Y 354.785,Z 222.42,A -85,B 0,C 180,E1 -19364.224,E2 -19364.224} C_VEL
LIN {X 0,Y 348.394,Z 218.079,A -85,B 0,C 180,E1 -19366.05,E2 -19366.05} C_VEL
LIN {X 0,Y 342.477,Z 213.774,A -85,B 0,C 180,E1 -19367.555,E2 -19367.555} C_VEL
LIN {X 0,Y 335.202,Z 208.652,A -85,B 0,C 180,E1 -19369.2,E2 -19369.2} C_VEL
LIN {X 0,Y 328.999,Z 203.917,A -85,B 0,C 180,E1 -19370.484,E2 -19370.484} C_VEL
LIN {X 0,Y 322.176,Z 198.715,A -85,B 0,C 180,E1 -19371.755,E2 -19371.755} C_VEL
LIN {X 0,Y 313.108,Z 191.534,A -85,B 0,C 180,E1 -19373.239,E2 -19373.239} C_VEL
LIN {X 0,Y 303.294,Z 183.295,A -85,B 0,C 180,E1 -19374.586,E2 -19374.586} C_VEL
LIN {X 0,Y 291.029,Z 172.23,A -85,B 0,C 180,E1 -19376.059,E2 -19376.059} C_VEL
LIN {X 0,Y 278.414,Z 159.223,A -85,B 0,C 180,E1 -19377.718,E2 -19377.718} C_VEL
LIN {X 0,Y 269.446,Z 148.237,A -85,B 0,C 180,E1 -19379.061,E2 -19379.061} C_VEL
LIN {X 0,Y 261.382,Z 136.111,A -85,B 0,C 180,E1 -19380.434,E2 -19380.434} C_VEL
LIN {X 0,Y 249.174,Z 113.172,A -85,B 0,C 180,E1 -19382.88,E2 -19382.88} C_VEL
LIN {X 0,Y 243.533,Z 103.381,A -85,B 0,C 180,E1 -19384.09,E2 -19384.09} C_VEL
LIN {X 0,Y 242.203,Z 100.716,A -85,B 0,C 180,E1 -19384.447,E2 -19384.447} C_VEL
LIN {X 0,Y 242.036,Z 99.889,A -85,B 0,C 180,E1 -19384.817,E2 -19384.817} C_VEL
LIN {X 0,Y 242.004,Z 99.838,A -85,B 0,C 180,E1 -19388.364,E2 -19388.364} C_VEL
LIN {X 0,Y 241.935,Z 99.785,A -85,B 0,C 180,E1 -19391.923,E2 -19391.923} C_VEL
LIN {X 0,Y 241.935,Z 99.849,A -85,B 0,C 180,E1 -19396.571,E2 -19396.571} C_VEL
LIN {X 0,Y 241.977,Z 99.827,A -85,B 0,C 180,E1 -19400.286,E2 -19400.286} C_VEL
LIN {X 0,Y 242.034,Z 99.816,A -85,B 0,C 180,E1 -19404.498,E2 -19404.498} C_VEL
LIN {X 0,Y 241.973,Z 99.844,A -85,B 0,C 180,E1 -19408.481,E2 -19408.481} C_VEL
LIN {X 0,Y 242,Z 99.809,A -85,B 0,C 180,E1 -19412.313,E2 -19412.313} C_VEL
LIN {X 0,Y 242.056,Z 99.832,A -85,B 0,C 180,E1 -19416.017,E2 -19416.017} C_VEL
LIN {X 0,Y 242.036,Z 99.805,A -85,B 0,C 180,E1 -19419.609,E2 -19419.609} C_VEL
LIN {X 0,Y 242.162,Z 99.802,A -85,B 0,C 180,E1 -19423.279,E2 -19423.279} C_VEL
LIN {X 0,Y 242.187,Z 99.789,A -85,B 0,C 180,E1 -19428.281,E2 -19428.281} C_VEL
LIN {X 0,Y 242.428,Z 99.753,A -85,B 0,C 180,E1 -19431.667,E2 -19431.667} C_VEL
LIN {X 0,Y 242.26,Z 99.807,A -85,B 0,C 180,E1 -19435.008,E2 -19435.008} C_VEL
LIN {X 0,Y 242.636,Z 99.726,A -85,B 0,C 180,E1 -19438.341,E2 -19438.341} C_VEL
LIN {X 0,Y 242.636,Z 99.729,A -85,B 0,C 180,E1 -19441.661,E2 -19441.661} C_VEL
LIN {X 0,Y 242.435,Z 99.775,A -85,B 0,C 180,E1 -19446.66,E2 -19446.66} C_VEL
LIN {X 0,Y 242.315,Z 99.756,A -85,B 0,C 180,E1 -19450.023,E2 -19450.023} C_VEL
LIN {X 0,Y 242.168,Z 99.815,A -85,B 0,C 180,E1 -19455.142,E2 -19455.142} C_VEL
LIN {X 0,Y 242.074,Z 99.788,A -85,B 0,C 180,E1 -19458.625,E2 -19458.625} C_VEL
LIN {X 0,Y 242.015,Z 99.834,A -85,B 0,C 180,E1 -19462.181,E2 -19462.181} C_VEL
LIN {X 0,Y 242.068,Z 99.804,A -85,B 0,C 180,E1 -19465.839,E2 -19465.839} C_VEL
LIN {X 0,Y 242.009,Z 99.831,A -85,B 0,C 180,E1 -19469.584,E2 -19469.584} C_VEL
LIN {X 0,Y 241.982,Z 99.818,A -85,B 0,C 180,E1 -19473.493,E2 -19473.493} C_VEL
LIN {X 0,Y 241.992,Z 99.842,A -85,B 0,C 180,E1 -19477.582,E2 -19477.582} C_VEL
LIN {X 0,Y 241.936,Z 99.845,A -85,B 0,C 180,E1 -19481.924,E2 -19481.924} C_VEL
LIN {X 0,Y 241.933,Z 99.85,A -85,B 0,C 180,E1 -19486.573,E2 -19486.573} C_VEL
LIN {X 0,Y 242.005,Z 99.936,A -85,B 0,C 180,E1 -19489.419,E2 -19489.419} C_VEL
LIN {X 0,Y 243.633,Z 106.743,A -85,B 0,C 180,E1 -19493.385,E2 -19493.385} C_VEL
LIN {X 0,Y 244.161,Z 109.654,A -85,B 0,C 180,E1 -19494.999,E2 -19494.999} C_VEL
LIN {X 0,Y 244.359,Z 111.634,A -85,B 0,C 180,E1 -19495.575,E2 -19495.575} C_VEL
LIN {X 0,Y 244.485,Z 114.477,A -85,B 0,C 180,E1 -19495.951,E2 -19495.951} C_VEL
LIN {X 0,Y 244.532,Z 118.347,A -85,B 0,C 180,E1 -19496.21,E2 -19496.21} C_VEL
LIN {X 0,Y 244.935,Z 126.896,A -85,B 0,C 180,E1 -19496.565,E2 -19496.565} C_VEL
LIN {X 0,Y 245.669,Z 129.509,A -85,B 0,C 180,E1 -19496.768,E2 -19496.768} C_VEL
LIN {X 0,Y 249.402,Z 138.614,A -85,B 0,C 180,E1 -19497.628,E2 -19497.628} C_VEL
LIN {X 0,Y 253.24,Z 159.35,A -85,B 0,C 180,E1 -19498.848,E2 -19498.848} C_VEL
LIN {X 0,Y 254.244,Z 166.745,A -85,B 0,C 180,E1 -19499.221,E2 -19499.221} C_VEL
LIN {X 0,Y 252.409,Z 217.245,A -85,B 0,C 180,E1 -19500.65,E2 -19500.65} C_VEL
LIN {X 0,Y 251.554,Z 227.722,A -85,B 0,C 180,E1 -19501.12,E2 -19501.12} C_VEL
LIN {X 0,Y 250.388,Z 237.401,A -85,B 0,C 180,E1 -19501.728,E2 -19501.728} C_VEL
LIN {X 0,Y 249.069,Z 246.473,A -85,B 0,C 180,E1 -19502.48,E2 -19502.48} C_VEL
LIN {X 0,Y 247.526,Z 255.604,A -85,B 0,C 180,E1 -19503.437,E2 -19503.437} C_VEL
LIN {X 0,Y 245.711,Z 264.595,A -85,B 0,C 180,E1 -19504.593,E2 -19504.593} C_VEL
LIN {X 0,Y 243.824,Z 273.321,A -85,B 0,C 180,E1 -19505.975,E2 -19505.975} C_VEL
LIN {X 0,Y 242.066,Z 280.712,A -85,B 0,C 180,E1 -19507.375,E2 -19507.375} C_VEL
LIN {X 0,Y 240.272,Z 287.929,A -85,B 0,C 180,E1 -19509.003,E2 -19509.003} C_VEL
LIN {X 0,Y 238.471,Z 295.509,A -85,B 0,C 180,E1 -19511.084,E2 -19511.084} C_VEL
LIN {X 0,Y 236.818,Z 301.826,A -85,B 0,C 180,E1 -19513.181,E2 -19513.181} C_VEL
LIN {X 0,Y 235.386,Z 307.085,A -85,B 0,C 180,E1 -19515.298,E2 -19515.298} C_VEL
LIN {X 0,Y 234.152,Z 312.217,A -85,B 0,C 180,E1 -19517.872,E2 -19517.872} C_VEL
LIN {X 0,Y 233.361,Z 316.209,A -85,B 0,C 180,E1 -19520.466,E2 -19520.466} C_VEL
LIN {X 0,Y 232.874,Z 319.162,A -85,B 0,C 180,E1 -19523.066,E2 -19523.066} C_VEL
LIN {X 0,Y 232.672,Z 321.615,A -85,B 0,C 180,E1 -19526.537,E2 -19526.537} C_VEL
LIN {X 0,Y 232.729,Z 322.208,A -85,B 0,C 180,E1 -19528.27,E2 -19528.27} C_VEL
LIN {X 0,Y 232.802,Z 322.365,A -85,B 0,C 180,E1 -19530,E2 -19530} C_VEL
LIN {X 0,Y 232.729,Z 322.208,A -85,B 0,C 180,E1 -19531.73,E2 -19531.73} C_VEL
LIN {X 0,Y 232.689,Z 320.937,A -85,B 0,C 180,E1 -19534.637,E2 -19534.637} C_VEL
LIN {X 0,Y 232.874,Z 319.162,A -85,B 0,C 180,E1 -19536.934,E2 -19536.934} C_VEL
LIN {X 0,Y 233.361,Z 316.209,A -85,B 0,C 180,E1 -19539.534,E2 -19539.534} C_VEL
LIN {X 0,Y 234.152,Z 312.217,A -85,B 0,C 180,E1 -19542.128,E2 -19542.128} C_VEL
LIN {X 0,Y 235.385,Z 307.085,A -85,B 0,C 180,E1 -19544.702,E2 -19544.702} C_VEL
LIN {X 0,Y 236.821,Z 301.826,A -85,B 0,C 180,E1 -19546.819,E2 -19546.819} C_VEL
LIN {X 0,Y 238.477,Z 295.51,A -85,B 0,C 180,E1 -19548.915,E2 -19548.915} C_VEL
LIN {X 0,Y 239.94,Z 289.558,A -85,B 0,C 180,E1 -19550.578,E2 -19550.578} C_VEL
LIN {X 0,Y 241.602,Z 282.631,A -85,B 0,C 180,E1 -19552.22,E2 -19552.22} C_VEL
LIN {X 0,Y 243.568,Z 274.455,A -85,B 0,C 180,E1 -19553.826,E2 -19553.826} C_VEL
LIN {X 0,Y 245.461,Z 265.947,A -85,B 0,C 180,E1 -19555.207,E2 -19555.207} C_VEL
LIN {X 0,Y 247.22,Z 257.235,A -85,B 0,C 180,E1 -19556.371,E2 -19556.371} C_VEL
LIN {X 0,Y 248.736,Z 248.486,A -85,B 0,C 180,E1 -19557.332,E2 -19557.332} C_VEL
LIN {X 0,Y 250.228,Z 238.689,A -85,B 0,C 180,E1 -19558.177,E2 -19558.177} C_VEL
LIN {X 0,Y 251.412,Z 228.548,A -85,B 0,C 180,E1 -19558.844,E2 -19558.844} C_VEL
LIN {X 0,Y 252.278,Z 218.477,A -85,B 0,C 180,E1 -19559.31,E2 -19559.31} C_VEL
LIN {X 0,Y 253.39,Z 189.757,A -85,B 0,C 180,E1 -19560.153,E2 -19560.153} C_VEL
LIN {X 0,Y 254.194,Z 165.185,A -85,B 0,C 180,E1 -19560.836,E2 -19560.836} C_VEL
LIN {X 0,Y 250.528,Z 144.229,A -85,B 0,C 180,E1 -19562.024,E2 -19562.024} C_VEL
LIN {X 0,Y 248.992,Z 137.274,A -85,B 0,C 180,E1 -19562.476,E2 -19562.476} C_VEL
LIN {X 0,Y 241.908,Z 121.143,A -85,B 0,C 180,E1 -19564.106,E2 -19564.106} C_VEL
LIN {X 0,Y 237.353,Z 111.527,A -85,B 0,C 180,E1 -19565.248,E2 -19565.248} C_VEL
LIN {X 0,Y 236.777,Z 108.562,A -85,B 0,C 180,E1 -19566.734,E2 -19566.734} C_VEL
LIN {X 0,Y 235.382,Z 102.661,A -85,B 0,C 180,E1 -19570.272,E2 -19570.272} C_VEL
LIN {X 0,Y 234.92,Z 100.722,A -85,B 0,C 180,E1 -19571.589,E2 -19571.589} C_VEL
LIN {X 0,Y 234.886,Z 100.717,A -85,B 0,C 180,E1 -19575.898,E2 -19575.898} C_VEL
LIN {X 0,Y 234.883,Z 100.713,A -85,B 0,C 180,E1 -19578.831,E2 -19578.831} C_VEL
LIN {X 0,Y 234.92,Z 100.71,A -85,B 0,C 180,E1 -19581.078,E2 -19581.078} C_VEL
LIN {X 0,Y 234.932,Z 100.694,A -85,B 0,C 180,E1 -19585.361,E2 -19585.361} C_VEL
LIN {X 0,Y 234.924,Z 100.722,A -85,B 0,C 180,E1 -19589.43,E2 -19589.43} C_VEL
LIN {X 0,Y 234.995,Z 100.681,A -85,B 0,C 180,E1 -19593.793,E2 -19593.793} C_VEL
LIN {X 0,Y 235.013,Z 100.69,A -85,B 0,C 180,E1 -19598.969,E2 -19598.969} C_VEL
LIN {X 0,Y 235.098,Z 100.671,A -85,B 0,C 180,E1 -19603.059,E2 -19603.059} C_VEL
LIN {X 0,Y 235.148,Z 100.671,A -85,B 0,C 180,E1 -19607.923,E2 -19607.923} C_VEL
LIN {X 0,Y 235.378,Z 100.624,A -85,B 0,C 180,E1 -19611.413,E2 -19611.413} C_VEL
LIN {X 0,Y 235.406,Z 100.646,A -85,B 0,C 180,E1 -19613.14,E2 -19613.14} C_VEL
LIN {X 0,Y 235.596,Z 100.605,A -85,B 0,C 180,E1 -19618.29,E2 -19618.29} C_VEL
LIN {X 0,Y 235.596,Z 100.603,A -85,B 0,C 180,E1 -19621.709,E2 -19621.709} C_VEL
LIN {X 0,Y 235.404,Z 100.649,A -85,B 0,C 180,E1 -19626.858,E2 -19626.858} C_VEL
LIN {X 0,Y 235.238,Z 100.639,A -85,B 0,C 180,E1 -19630.326,E2 -19630.326} C_VEL
LIN {X 0,Y 235.113,Z 100.694,A -85,B 0,C 180,E1 -19635.605,E2 -19635.605} C_VEL
LIN {X 0,Y 235.007,Z 100.671,A -85,B 0,C 180,E1 -19639.205,E2 -19639.205} C_VEL
LIN {X 0,Y 234.96,Z 100.717,A -85,B 0,C 180,E1 -19642.882,E2 -19642.882} C_VEL
LIN {X 0,Y 234.966,Z 100.685,A -85,B 0,C 180,E1 -19646.657,E2 -19646.657} C_VEL
LIN {X 0,Y 234.921,Z 100.722,A -85,B 0,C 180,E1 -19650.568,E2 -19650.568} C_VEL
LIN {X 0,Y 234.958,Z 100.692,A -85,B 0,C 180,E1 -19654.632,E2 -19654.632} C_VEL
LIN {X 0,Y 234.939,Z 100.712,A -85,B 0,C 180,E1 -19658.944,E2 -19658.944} C_VEL
LIN {X 0,Y 234.913,Z 100.724,A -85,B 0,C 180,E1 -19663.479,E2 -19663.479} C_VEL
LIN {X 0,Y 234.877,Z 100.671,A -85,B 0,C 180,E1 -19666.512,E2 -19666.512} C_VEL
LIN {X 0,Y 234.952,Z 100.698,A -85,B 0,C 180,E1 -19671.085,E2 -19671.085} C_VEL
LIN {X 0,Y 235.007,Z 100.923,A -85,B 0,C 180,E1 -19674.156,E2 -19674.156} C_VEL
LIN {X 0,Y 235.253,Z 101.911,A -85,B 0,C 180,E1 -19674.446,E2 -19674.446} C_VEL
LIN {X 0,Y 236.913,Z 104.755,A -85,B 0,C 180,E1 -19674.861,E2 -19674.861} C_VEL
LIN {X 0,Y 246.832,Z 122.294,A -85,B 0,C 180,E1 -19677.076,E2 -19677.076} C_VEL
LIN {X 0,Y 256.869,Z 141.436,A -85,B 0,C 180,E1 -19679.139,E2 -19679.139} C_VEL
LIN {X 0,Y 265.912,Z 154.803,A -85,B 0,C 180,E1 -19680.712,E2 -19680.712} C_VEL
LIN {X 0,Y 276.734,Z 167.51,A -85,B 0,C 180,E1 -19682.336,E2 -19682.336} C_VEL
LIN {X 0,Y 290.947,Z 181.718,A -85,B 0,C 180,E1 -19684.188,E2 -19684.188} C_VEL
LIN {X 0,Y 302.509,Z 191.638,A -85,B 0,C 180,E1 -19685.561,E2 -19685.561} C_VEL
LIN {X 0,Y 311.973,Z 199.402,A -85,B 0,C 180,E1 -19686.838,E2 -19686.838} C_VEL
LIN {X 0,Y 319.806,Z 205.499,A -85,B 0,C 180,E1 -19688.1,E2 -19688.1} C_VEL
LIN {X 0,Y 327.486,Z 211.195,A -85,B 0,C 180,E1 -19689.523,E2 -19689.523} C_VEL
LIN {X 0,Y 335.859,Z 217.51,A -85,B 0,C 180,E1 -19691.288,E2 -19691.288} C_VEL
LIN {X 0,Y 343.78,Z 222.931,A -85,B 0,C 180,E1 -19693.166,E2 -19693.166} C_VEL
LIN {X 0,Y 350.168,Z 227.585,A -85,B 0,C 180,E1 -19694.92,E2 -19694.92} C_VEL
LIN {X 0,Y 355.827,Z 230.997,A -85,B 0,C 180,E1 -19696.646,E2 -19696.646} C_VEL
LIN {X 0,Y 359.309,Z 233.14,A -85,B 0,C 180,E1 -19697.852,E2 -19697.852} C_VEL
LIN {X 0,Y 363.946,Z 236.637,A -85,B 0,C 180,E1 -19699.771,E2 -19699.771} C_VEL
LIN {X 0,Y 366.909,Z 238.505,A -85,B 0,C 180,E1 -19701.185,E2 -19701.185} C_VEL
LIN {X 0,Y 369.056,Z 239.672,A -85,B 0,C 180,E1 -19702.34,E2 -19702.34} C_VEL
LIN {X 0,Y 370.853,Z 240.586,A -85,B 0,C 180,E1 -19703.471,E2 -19703.471} C_VEL
LIN {X 0,Y 372.383,Z 241.214,A -85,B 0,C 180,E1 -19704.585,E2 -19704.585} C_VEL
LIN {X 0,Y 373.613,Z 241.726,A -85,B 0,C 180,E1 -19705.685,E2 -19705.685} C_VEL
LIN {X 0,Y 374.608,Z 241.955,A -85,B 0,C 180,E1 -19706.774,E2 -19706.774} C_VEL
LIN {X 0,Y 375.244,Z 242.315,A -85,B 0,C 180,E1 -19707.853,E2 -19707.853} C_VEL
LIN {X 0,Y 375.591,Z 242.631,A -85,B 0,C 180,E1 -19708.928,E2 -19708.928} C_VEL
LIN {X 0,Y 375.776,Z 242.521,A -85,B 0,C 180,E1 -19710,E2 -19710} C_VEL
LIN {X 0,Y 375.629,Z 242.519,A -85,B 0,C 180,E1 -19711.072,E2 -19711.072} C_VEL
LIN {X 0,Y 375.258,Z 242.288,A -85,B 0,C 180,E1 -19712.147,E2 -19712.147} C_VEL
LIN {X 0,Y 374.622,Z 241.939,A -85,B 0,C 180,E1 -19713.226,E2 -19713.226} C_VEL
LIN {X 0,Y 373.577,Z 241.639,A -85,B 0,C 180,E1 -19714.394,E2 -19714.394} C_VEL
LIN {X 0,Y 372.394,Z 241.249,A -85,B 0,C 180,E1 -19715.415,E2 -19715.415} C_VEL
LIN {X 0,Y 370.877,Z 240.576,A -85,B 0,C 180,E1 -19716.529,E2 -19716.529} C_VEL
LIN {X 0,Y 368.833,Z 239.58,A -85,B 0,C 180,E1 -19717.764,E2 -19717.764} C_VEL
LIN {X 0,Y 365.347,Z 237.552,A -85,B 0,C 180,E1 -19719.585,E2 -19719.585} C_VEL
LIN {X 0,Y 361.044,Z 234.544,A -85,B 0,C 180,E1 -19721.454,E2 -19721.454} C_VEL
LIN {X 0,Y 357.317,Z 231.811,A -85,B 0,C 180,E1 -19722.854,E2 -19722.854} C_VEL
LIN {X 0,Y 351.866,Z 228.642,A -85,B 0,C 180,E1 -19724.58,E2 -19724.58} C_VEL
LIN {X 0,Y 345.694,Z 224.436,A -85,B 0,C 180,E1 -19726.317,E2 -19726.317} C_VEL
LIN {X 0,Y 340.506,Z 220.633,A -85,B 0,C 180,E1 -19727.641,E2 -19727.641} C_VEL
LIN {X 0,Y 333.065,Z 215.487,A -85,B 0,C 180,E1 -19729.32,E2 -19729.32} C_VEL
LIN {X 0,Y 326.218,Z 210.298,A -85,B 0,C 180,E1 -19730.721,E2 -19730.721} C_VEL
LIN {X 0,Y 318.784,Z 204.676,A -85,B 0,C 180,E1 -19732.077,E2 -19732.077} C_VEL
LIN {X 0,Y 310.886,Z 198.588,A -85,B 0,C 180,E1 -19733.311,E2 -19733.311} C_VEL
LIN {X 0,Y 302.321,Z 191.535,A -85,B 0,C 180,E1 -19734.461,E2 -19734.461} C_VEL
LIN {X 0,Y 289.143,Z 180.076,A -85,B 0,C 180,E1 -19736.031,E2 -19736.031} C_VEL
LIN {X 0,Y 274.782,Z 165.416,A -85,B 0,C 180,E1 -19737.94,E2 -19737.94} C_VEL
LIN {X 0,Y 264.882,Z 153.388,A -85,B 0,C 180,E1 -19739.458,E2 -19739.458} C_VEL
LIN {X 0,Y 256.36,Z 140.57,A -85,B 0,C 180,E1 -19740.958,E2 -19740.958} C_VEL
LIN {X 0,Y 243.898,Z 116.93,A -85,B 0,C 180,E1 -19743.56,E2 -19743.56} C_VEL
LIN {X 0,Y 236.564,Z 104.341,A -85,B 0,C 180,E1 -19745.214,E2 -19745.214} C_VEL
LIN {X 0,Y 235.131,Z 101.421,A -85,B 0,C 180,E1 -19745.648,E2 -19745.648} C_VEL
LIN {X 0,Y 234.953,Z 100.73,A -85,B 0,C 180,E1 -19746.136,E2 -19746.136} C_VEL
LIN {X 0,Y 234.939,Z 100.699,A -85,B 0,C 180,E1 -19748.945,E2 -19748.945} C_VEL
LIN {X 0,Y 234.877,Z 100.671,A -85,B 0,C 180,E1 -19753.488,E2 -19753.488} C_VEL
LIN {X 0,Y 234.913,Z 100.724,A -85,B 0,C 180,E1 -19756.521,E2 -19756.521} C_VEL
LIN {X 0,Y 234.952,Z 100.711,A -85,B 0,C 180,E1 -19761.087,E2 -19761.087} C_VEL
LIN {X 0,Y 234.958,Z 100.692,A -85,B 0,C 180,E1 -19765.368,E2 -19765.368} C_VEL
LIN {X 0,Y 234.921,Z 100.722,A -85,B 0,C 180,E1 -19769.432,E2 -19769.432} C_VEL
LIN {X 0,Y 234.992,Z 100.685,A -85,B 0,C 180,E1 -19773.795,E2 -19773.795} C_VEL
LIN {X 0,Y 235.01,Z 100.689,A -85,B 0,C 180,E1 -19778.971,E2 -19778.971} C_VEL
LIN {X 0,Y 235.095,Z 100.678,A -85,B 0,C 180,E1 -19783.06,E2 -19783.06} C_VEL
LIN {X 0,Y 235.147,Z 100.671,A -85,B 0,C 180,E1 -19787.925,E2 -19787.925} C_VEL
LIN {X 0,Y 235.377,Z 100.627,A -85,B 0,C 180,E1 -19791.415,E2 -19791.415} C_VEL
LIN {X 0,Y 235.404,Z 100.649,A -85,B 0,C 180,E1 -19793.142,E2 -19793.142} C_VEL
LIN {X 0,Y 235.596,Z 100.603,A -85,B 0,C 180,E1 -19798.291,E2 -19798.291} C_VEL
LIN {X 0,Y 235.596,Z 100.605,A -85,B 0,C 180,E1 -19801.71,E2 -19801.71} C_VEL
LIN {X 0,Y 235.406,Z 100.646,A -85,B 0,C 180,E1 -19806.86,E2 -19806.86} C_VEL
LIN {X 0,Y 235.239,Z 100.637,A -85,B 0,C 180,E1 -19810.327,E2 -19810.327} C_VEL
LIN {X 0,Y 235.115,Z 100.688,A -85,B 0,C 180,E1 -19815.607,E2 -19815.607} C_VEL
LIN {X 0,Y 235.01,Z 100.668,A -85,B 0,C 180,E1 -19819.206,E2 -19819.206} C_VEL
LIN {X 0,Y 234.963,Z 100.715,A -85,B 0,C 180,E1 -19822.884,E2 -19822.884} C_VEL
LIN {X 0,Y 234.969,Z 100.682,A -85,B 0,C 180,E1 -19826.658,E2 -19826.658} C_VEL
LIN {X 0,Y 234.924,Z 100.722,A -85,B 0,C 180,E1 -19830.57,E2 -19830.57} C_VEL
LIN {X 0,Y 234.932,Z 100.694,A -85,B 0,C 180,E1 -19834.639,E2 -19834.639} C_VEL
LIN {X 0,Y 234.944,Z 100.707,A -85,B 0,C 180,E1 -19838.945,E2 -19838.945} C_VEL
LIN {X 0,Y 234.881,Z 100.722,A -85,B 0,C 180,E1 -19843.489,E2 -19843.489} C_VEL
LIN {X 0,Y 234.885,Z 100.727,A -85,B 0,C 180,E1 -19846.514,E2 -19846.514} C_VEL
LIN {X 0,Y 234.909,Z 100.803,A -85,B 0,C 180,E1 -19848.559,E2 -19848.559} C_VEL
LIN {X 0,Y 236.491,Z 107.139,A -85,B 0,C 180,E1 -19852.431,E2 -19852.431} C_VEL
LIN {X 0,Y 237.319,Z 111.286,A -85,B 0,C 180,E1 -19854.703,E2 -19854.703} C_VEL
LIN {X 0,Y 239.041,Z 115.193,A -85,B 0,C 180,E1 -19855.219,E2 -19855.219} C_VEL
LIN {X 0,Y 245.669,Z 129.509,A -85,B 0,C 180,E1 -19856.768,E2 -19856.768} C_VEL
LIN {X 0,Y 246.777,Z 133.062,A -85,B 0,C 180,E1 -19857.056,E2 -19857.056} C_VEL
LIN {X 0,Y 247.339,Z 136.849,A -85,B 0,C 180,E1 -19857.268,E2 -19857.268} C_VEL
LIN {X 0,Y 247.39,Z 144.715,A -85,B 0,C 180,E1 -19857.54,E2 -19857.54} C_VEL
LIN {X 0,Y 246.916,Z 156.821,A -85,B 0,C 180,E1 -19857.878,E2 -19857.878} C_VEL
LIN {X 0,Y 247.22,Z 160.789,A -85,B 0,C 180,E1 -19858.055,E2 -19858.055} C_VEL
LIN {X 0,Y 248.138,Z 166.926,A -85,B 0,C 180,E1 -19858.39,E2 -19858.39} C_VEL
LIN {X 0,Y 246.206,Z 217.71,A -85,B 0,C 180,E1 -19859.866,E2 -19859.866} C_VEL
LIN {X 0,Y 245.26,Z 228.528,A -85,B 0,C 180,E1 -19860.373,E2 -19860.373} C_VEL
LIN {X 0,Y 243.791,Z 239.785,A -85,B 0,C 180,E1 -19861.127,E2 -19861.127} C_VEL
LIN {X 0,Y 241.782,Z 252.148,A -85,B 0,C 180,E1 -19862.285,E2 -19862.285} C_VEL
LIN {X 0,Y 239.611,Z 263.054,A -85,B 0,C 180,E1 -19863.664,E2 -19863.664} C_VEL
LIN {X 0,Y 237.582,Z 271.995,A -85,B 0,C 180,E1 -19865.069,E2 -19865.069} C_VEL
LIN {X 0,Y 235.506,Z 280.521,A -85,B 0,C 180,E1 -19866.709,E2 -19866.709} C_VEL
LIN {X 0,Y 233.635,Z 287.738,A -85,B 0,C 180,E1 -19868.377,E2 -19868.377} C_VEL
LIN {X 0,Y 232.195,Z 293.543,A -85,B 0,C 180,E1 -19869.958,E2 -19869.958} C_VEL
LIN {X 0,Y 230.256,Z 300.477,A -85,B 0,C 180,E1 -19872.228,E2 -19872.228} C_VEL
LIN {X 0,Y 229.073,Z 304.979,A -85,B 0,C 180,E1 -19873.971,E2 -19873.971} C_VEL
LIN {X 0,Y 227.515,Z 310.469,A -85,B 0,C 180,E1 -19876.604,E2 -19876.604} C_VEL
LIN {X 0,Y 226.57,Z 314.799,A -85,B 0,C 180,E1 -19879.274,E2 -19879.274} C_VEL
LIN {X 0,Y 226.134,Z 317.17,A -85,B 0,C 180,E1 -19881.06,E2 -19881.06} C_VEL
LIN {X 0,Y 225.811,Z 318.971,A -85,B 0,C 180,E1 -19882.849,E2 -19882.849} C_VEL
LIN {X 0,Y 225.586,Z 321.425,A -85,B 0,C 180,E1 -19886.428,E2 -19886.428} C_VEL
LIN {X 0,Y 225.625,Z 322.018,A -85,B 0,C 180,E1 -19888.215,E2 -19888.215} C_VEL
LIN {X 0,Y 225.714,Z 322.175,A -85,B 0,C 180,E1 -19890,E2 -19890} C_VEL
LIN {X 0,Y 225.624,Z 322.018,A -85,B 0,C 180,E1 -19891.785,E2 -19891.785} C_VEL
LIN {X 0,Y 225.587,Z 320.951,A -85,B 0,C 180,E1 -19894.475,E2 -19894.475} C_VEL
LIN {X 0,Y 225.811,Z 318.971,A -85,B 0,C 180,E1 -19897.151,E2 -19897.151} C_VEL
LIN {X 0,Y 226.326,Z 316.017,A -85,B 0,C 180,E1 -19899.834,E2 -19899.834} C_VEL
LIN {X 0,Y 227.16,Z 312.025,A -85,B 0,C 180,E1 -19902.508,E2 -19902.508} C_VEL
LIN {X 0,Y 228.506,Z 306.894,A -85,B 0,C 180,E1 -19905.155,E2 -19905.155} C_VEL
LIN {X 0,Y 229.979,Z 301.634,A -85,B 0,C 180,E1 -19907.335,E2 -19907.335} C_VEL
LIN {X 0,Y 231.749,Z 295.318,A -85,B 0,C 180,E1 -19909.486,E2 -19909.486} C_VEL
LIN {X 0,Y 233.277,Z 289.366,A -85,B 0,C 180,E1 -19911.194,E2 -19911.194} C_VEL
LIN {X 0,Y 235.025,Z 282.439,A -85,B 0,C 180,E1 -19912.876,E2 -19912.876} C_VEL
LIN {X 0,Y 237.095,Z 274.265,A -85,B 0,C 180,E1 -19914.519,E2 -19914.519} C_VEL
LIN {X 0,Y 239.052,Z 265.756,A -85,B 0,C 180,E1 -19915.933,E2 -19915.933} C_VEL
LIN {X 0,Y 240.883,Z 257.045,A -85,B 0,C 180,E1 -19917.121,E2 -19917.121} C_VEL
LIN {X 0,Y 242.454,Z 248.296,A -85,B 0,C 180,E1 -19918.102,E2 -19918.102} C_VEL
LIN {X 0,Y 244,Z 238.499,A -85,B 0,C 180,E1 -19918.964,E2 -19918.964} C_VEL
LIN {X 0,Y 245.201,Z 228.554,A -85,B 0,C 180,E1 -19919.633,E2 -19919.633} C_VEL
LIN {X 0,Y 246.159,Z 217.765,A -85,B 0,C 180,E1 -19920.136,E2 -19920.136} C_VEL
LIN {X 0,Y 247.82,Z 175.847,A -85,B 0,C 180,E1 -19921.358,E2 -19921.358} C_VEL
LIN {X 0,Y 248.126,Z 166.416,A -85,B 0,C 180,E1 -19921.629,E2 -19921.629} C_VEL
LIN {X 0,Y 244.219,Z 143.898,A -85,B 0,C 180,E1 -19922.959,E2 -19922.959} C_VEL
LIN {X 0,Y 243.13,Z 139.69,A -85,B 0,C 180,E1 -19923.269,E2 -19923.269} C_VEL
LIN {X 0,Y 235.991,Z 123.368,A -85,B 0,C 180,E1 -19924.996,E2 -19924.996} C_VEL
LIN {X 0,Y 231.322,Z 114.127,A -85,B 0,C 180,E1 -19926.151,E2 -19926.151} C_VEL
LIN {X 0,Y 230.065,Z 111.026,A -85,B 0,C 180,E1 -19926.597,E2 -19926.597} C_VEL
LIN {X 0,Y 228.673,Z 104.995,A -85,B 0,C 180,E1 -19930.196,E2 -19930.196} C_VEL
LIN {X 0,Y 227.843,Z 101.667,A -85,B 0,C 180,E1 -19932.415,E2 -19932.415} C_VEL
LIN {X 0,Y 227.828,Z 101.594,A -85,B 0,C 180,E1 -19935.194,E2 -19935.194} C_VEL
LIN {X 0,Y 227.827,Z 101.587,A -85,B 0,C 180,E1 -19939.622,E2 -19939.622} C_VEL
LIN {X 0,Y 227.883,Z 101.582,A -85,B 0,C 180,E1 -19944.128,E2 -19944.128} C_VEL
LIN {X 0,Y 227.869,Z 101.598,A -85,B 0,C 180,E1 -19948.377,E2 -19948.377} C_VEL
LIN {X 0,Y 227.881,Z 101.565,A -85,B 0,C 180,E1 -19952.443,E2 -19952.443} C_VEL
LIN {X 0,Y 227.916,Z 101.591,A -85,B 0,C 180,E1 -19956.367,E2 -19956.367} C_VEL
LIN {X 0,Y 227.944,Z 101.551,A -85,B 0,C 180,E1 -19960.174,E2 -19960.174} C_VEL
